REGION Network 9: DataIn - Sollevatore 3
   RUNG wire#powerrail
      "ValveMachine_PB_Connector"(Enable := wire#w1, HMI_PB := "A03_HMI".MB3.Button.A0302.Centratori.Sollevamento, LB_PB_Rest := FALSE, LB_PB_Work := FALSE, LB_PB_StartStop := FALSE, Other_PB := "A03_HMI".MB3.Button.PB_Empty.Valve, PB => "A0302_Centratori".Sollevamento[3].DataIn.PB)
   END_RUNG
   RUNG wire#powerrail
      Contact( "A0302_Centratori".HMI.Selection.Sollevamento[3] )
   END_RUNG wire#w1
   RUNG wire#powerrail
      Contact( "A0302_Centratori_Centraggio_3_Testa_Ls_Basso" )
      Coil( "A0302_Centratori".Sollevamento[3].DataIn.Rest_Ls[1] )
   END_RUNG
   RUNG wire#powerrail
      Contact( "A0302_Centratori_Centraggio_3_Testa_Ls_Alto" )
      Coil( "A0302_Centratori".Sollevamento[3].DataIn.Work_Ls[1] )
   END_RUNG
   // the same network as SCL:
   "ValveMachine_PB_Connector"(Enable := "A0302_Centratori".HMI.Selection.Sollevamento[3],
                           HMI_PB := "A03_HMI".MB3.Button.A0302.Centratori.Sollevamento,
                           LB_PB_Rest := FALSE,
                           LB_PB_Work := FALSE,
                           LB_PB_StartStop := FALSE,
                           Other_PB := "A03_HMI".MB3.Button.PB_Empty.Valve,
                           PB => "A0302_Centratori".Sollevamento[3].DataIn.PB);
   "A0302_Centratori".Sollevamento[3].DataIn.Rest_Ls[1] := "A0302_Centratori_Centraggio_3_Testa_Ls_Basso";
   "A0302_Centratori".Sollevamento[3].DataIn.Work_Ls[1] := "A0302_Centratori_Centraggio_3_Testa_Ls_Alto";
END_REGION

REGION Network 11 (SCL): DSI
   // Di solito facciamo struct DSI con dentro Centratori

   "A0302_Centratori".DSI := "F_DB".DSI_V_Air_A0302_A0303;
END_REGION

REGION Network 12: [Centratori] - Machine Call
   RUNG wire#powerrail
      "A0302_Centratori"(AreaInterface := "Area03".AreaInterface, ZSI := "F_DB".ZSI_Zone25, DSI :=, DataIn :=, CIn :=, Config := "PrjConfig_A03".A0302.Centratori, MachineInterface =>, COut =>)
   END_RUNG
   // the same network as SCL:
   "A0302_Centratori"(AreaInterface := "Area03".AreaInterface,   // "A0302_Centratori_FB"
                      ZSI := "F_DB".ZSI_Zone25,
                      Config := "PrjConfig_A03".A0302.Centratori);
END_REGION

REGION Network 14: <<< DATA OUT >>>
END_REGION

REGION Network 15: DataOut - Centraggio 1
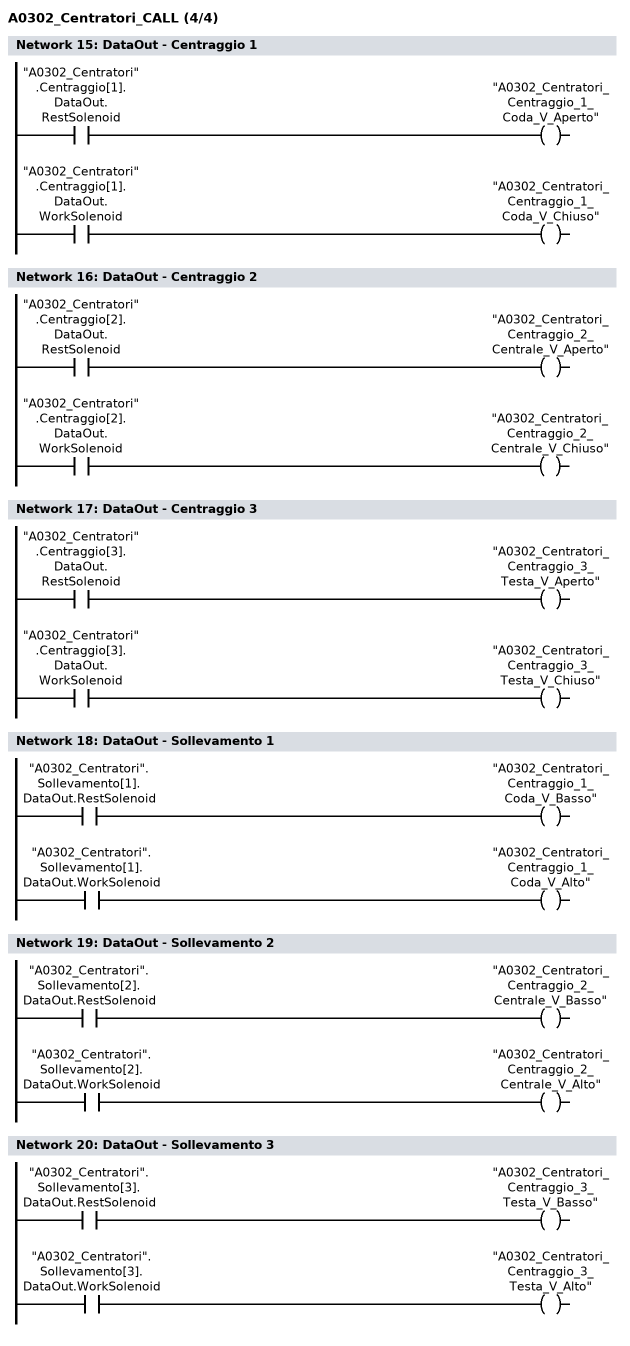
   RUNG wire#powerrail
      Contact( "A0302_Centratori".Centraggio[1].DataOut.RestSolenoid )
      Coil( "A0302_Centratori_Centraggio_1_Coda_V_Aperto" )
   END_RUNG
   RUNG wire#powerrail
      Contact( "A0302_Centratori".Centraggio[1].DataOut.WorkSolenoid )
      Coil( "A0302_Centratori_Centraggio_1_Coda_V_Chiuso" )
   END_RUNG
   // the same network as SCL:
   "A0302_Centratori_Centraggio_1_Coda_V_Aperto" := "A0302_Centratori".Centraggio[1].DataOut.RestSolenoid;
   "A0302_Centratori_Centraggio_1_Coda_V_Chiuso" := "A0302_Centratori".Centraggio[1].DataOut.WorkSolenoid;
END_REGION

REGION Network 16: DataOut - Centraggio 2
   RUNG wire#powerrail
      Contact( "A0302_Centratori".Centraggio[2].DataOut.RestSolenoid )
      Coil( "A0302_Centratori_Centraggio_2_Centrale_V_Aperto" )
   END_RUNG
   RUNG wire#powerrail
      Contact( "A0302_Centratori".Centraggio[2].DataOut.WorkSolenoid )
      Coil( "A0302_Centratori_Centraggio_2_Centrale_V_Chiuso" )
   END_RUNG
   // the same network as SCL:
   "A0302_Centratori_Centraggio_2_Centrale_V_Aperto" := "A0302_Centratori".Centraggio[2].DataOut.RestSolenoid;
   "A0302_Centratori_Centraggio_2_Centrale_V_Chiuso" := "A0302_Centratori".Centraggio[2].DataOut.WorkSolenoid;
END_REGION

REGION Network 17: DataOut - Centraggio 3
   RUNG wire#powerrail
      Contact( "A0302_Centratori".Centraggio[3].DataOut.RestSolenoid )
      Coil( "A0302_Centratori_Centraggio_3_Testa_V_Aperto" )
   END_RUNG
   RUNG wire#powerrail
      Contact( "A0302_Centratori".Centraggio[3].DataOut.WorkSolenoid )
      Coil( "A0302_Centratori_Centraggio_3_Testa_V_Chiuso" )
   END_RUNG
   // the same network as SCL:
   "A0302_Centratori_Centraggio_3_Testa_V_Aperto" := "A0302_Centratori".Centraggio[3].DataOut.RestSolenoid;
   "A0302_Centratori_Centraggio_3_Testa_V_Chiuso" := "A0302_Centratori".Centraggio[3].DataOut.WorkSolenoid;
END_REGION

REGION Network 18: DataOut - Sollevamento 1
   RUNG wire#powerrail
      Contact( "A0302_Centratori".Sollevamento[1].DataOut.RestSolenoid )
      Coil( "A0302_Centratori_Centraggio_1_Coda_V_Basso" )
   END_RUNG
   RUNG wire#powerrail
      Contact( "A0302_Centratori".Sollevamento[1].DataOut.WorkSolenoid )
      Coil( "A0302_Centratori_Centraggio_1_Coda_V_Alto" )
   END_RUNG
   // the same network as SCL:
   "A0302_Centratori_Centraggio_1_Coda_V_Basso" := "A0302_Centratori".Sollevamento[1].DataOut.RestSolenoid;
   "A0302_Centratori_Centraggio_1_Coda_V_Alto" := "A0302_Centratori".Sollevamento[1].DataOut.WorkSolenoid;
END_REGION

REGION Network 19: DataOut - Sollevamento 2
   RUNG wire#powerrail
      Contact( "A0302_Centratori".Sollevamento[2].DataOut.RestSolenoid )
      Coil( "A0302_Centratori_Centraggio_2_Centrale_V_Basso" )
   END_RUNG
   RUNG wire#powerrail
      Contact( "A0302_Centratori".Sollevamento[2].DataOut.WorkSolenoid )
      Coil( "A0302_Centratori_Centraggio_2_Centrale_V_Alto" )
   END_RUNG
   // the same network as SCL:
   "A0302_Centratori_Centraggio_2_Centrale_V_Basso" := "A0302_Centratori".Sollevamento[2].DataOut.RestSolenoid;
   "A0302_Centratori_Centraggio_2_Centrale_V_Alto" := "A0302_Centratori".Sollevamento[2].DataOut.WorkSolenoid;
END_REGION

REGION Network 20: DataOut - Sollevamento 3
   RUNG wire#powerrail
      Contact( "A0302_Centratori".Sollevamento[3].DataOut.RestSolenoid )
      Coil( "A0302_Centratori_Centraggio_3_Testa_V_Basso" )
   END_RUNG
   RUNG wire#powerrail
      Contact( "A0302_Centratori".Sollevamento[3].DataOut.WorkSolenoid )
      Coil( "A0302_Centratori_Centraggio_3_Testa_V_Alto" )
   END_RUNG
   // the same network as SCL:
   "A0302_Centratori_Centraggio_3_Testa_V_Basso" := "A0302_Centratori".Sollevamento[3].DataOut.RestSolenoid;
   "A0302_Centratori_Centraggio_3_Testa_V_Alto" := "A0302_Centratori".Sollevamento[3].DataOut.WorkSolenoid;
END_REGION
END_FUNCTION

FUNCTION_BLOCK "A0302_Centratori_FB"   // FB92, LAD
TITLE = <<< GESTIONE CENTRATORI >>>
// stored: MemoryReserve 100, SetENOAutomatically false
   VAR_INPUT
      AreaInterface : "AreaInterface";
      ZSI : "udt_ZoneSafetyInterface";
      DSI : "udt_DeviceSafetyInterface";
      DataIn : Struct
         OP : "OP_PB";
      END_STRUCT;
      CIn : Struct
         Manager : Struct
            Sollevamento : "ValveMachine_Manager";
            Centraggio : "ValveMachine_Manager";
         END_STRUCT;
         SemiAut_Pb : Bool;
         Rulliera : Struct
            Coda : Struct
               Sens : Struct
                  FTC_Rall : Bool;   // Sensori presenza materiale banco rallentamento ingresso
                  FTC_Prox_Ing : Bool;   // Sensori presenza materiale banco limite ingresso
               END_STRUCT;
            END_STRUCT;
            Centro : Struct
               Sens : Struct
                  FTC_Centrale : Bool;   // 2010BF1 - I50.2
               END_STRUCT;
            END_STRUCT;
         END_STRUCT;
         CarroPareggCoda : Struct
            Ax : "Positioning_DOL_Machine_COut";
            Bloccaggio : "ValveMachine_COut";
            BattutaVerticale : "ValveMachine_COut";
            PareggiatoreLong : "ValveMachine_COut";
            Sens : Struct
               FTC_Ingombro_In : Bool;   // 2012BF1 - I50.0
               FTC_Ingombro_Out : Bool;   // 2012BF2 - I50.1
               PresenzaMat : Bool;   // FC presenza materiale agganciato lato paregg coda
            END_STRUCT;
         END_STRUCT;
         CarroPareggTesta : Struct
            Ax : "Positioning_DOL_Machine_COut";
            Bloccaggio : "ValveMachine_COut";
            Centraggio : "ValveMachine_COut";
            Sollevatore : "ValveMachine_COut";
            Sens : Struct
               FTC1_Rall : Bool;   // 2010BF2 - I50.3
               FTC2_Prox_Ls : Bool;   // 2010BF3 - I50.4
               PresenzaMat : Bool;   // FC presenza materiale agganciato lato paregg testa
            END_STRUCT;
         END_STRUCT;
         BTrk : Struct
            ZoneA0302Entry_Empty : Bool;
            ZoneA0302Exit_Empty : Bool;
         END_STRUCT;
      END_STRUCT;
      Config : Struct
         Centraggio : Array[1..3] of "ValveMachine_Config";
         Sollevamento : Array[1..3] of "ValveMachine_Config";
         DelayMissingCondition : Time;
         WorkWindows : Struct   // Finestre di disattivazione Centratore 1 e 3 in funzione dei Carri
            Coda : Struct
               Min : LReal;
               Max : LReal;
            END_STRUCT;
            Testa : Struct
               Min : LReal;
               Max : LReal;
            END_STRUCT;
         END_STRUCT;
      END_STRUCT;
   END_VAR
   VAR_OUTPUT
      MachineInterface : "MachineInterface";
      COut : Struct
         Centratori : "ValveMachine_COut";
         Centraggio : "ValveMachine_COut";
         Sollevamento : "ValveMachine_COut";
      END_STRUCT;
   END_VAR
   VAR
      Alarm : Struct
         Centraggio : Array[1..3] of "ValveAlr";
         Sollevamento : Array[1..3] of "ValveAlr";
      END_STRUCT;
      Warning : Struct
         Centratore : Array[1..3] of "ValveMachine_Wng";
         Sollevamento : Array[1..3] of "ValveMachine_Wng";
         OP_REST_Centr_MissingCnd : Bool;   // Mancanza comando arresto
         OP_WORK_Centr_MissingCnd : Bool;   // Mancanza consenso lavoro
         OP_REST_Sollev_MissingCnd : Bool;   // Mancanza comando arresto
         OP_WORK_Sollev_MissingCnd : Bool;   // Mancanza consenso lavoro
      END_STRUCT;
      HMI : Struct
         Selection : Struct   // 0=Disable / 1=Enable Pin
            Centraggio : Array[1..3] of Bool;
            Sollevamento : Array[1..3] of Bool;
         END_STRUCT;
         Centratori_Sts : "UDT_HMI-Sts_ValvePosA0301";
         Centraggio_Sts { S7_SetPoint := 'True'} : "UDT_HMI-Sts_ValvePosA0301";
         Sollevamento_Sts { S7_SetPoint := 'True'} : "UDT_HMI-Sts_ValvePosA0301";
      END_STRUCT;
      Centraggio : Array[1..3] of "ValveMachine_FB";
      Sollevamento { S7_SetPoint := 'True'} : Array[1..3] of "ValveMachine_FB";
      Sts : Struct
         Centraggio : Struct
            OP_Rest_Cnd : Bool;
            Op_Work_Cnd : Bool;
         END_STRUCT;
         Sollevamento : Struct
            OP_Rest_Cnd : Bool;
            Op_Work_Cnd : Bool;
         END_STRUCT;
         Centratori_Alarm : Bool;
         Centraggio_AlarmPresence : Bool;
         Sollevamento_AlarmPresence : Bool;
         OP_CanMoveFreely : Bool;
      END_STRUCT;
      Ctrl : Struct
         Centraggio : Struct
            OP_Rest_Man : Bool;
            OP_Work_Man : Bool;
            OP_Rest_Aut : Bool;
            OP_Work_Aut : Bool;
            OP_Rest : Bool;
            OP_Work : Bool;
         END_STRUCT;
         Sollevamento : Struct
            OP_Rest_Man : Bool;
            OP_Work_Man : Bool;
            OP_Rest_Aut : Bool;
            OP_Work_Aut : Bool;
            OP_Rest : Bool;
            OP_Work : Bool;
         END_STRUCT;
      END_STRUCT;
      AUX : Struct
         Centraggio : Struct
            OP_Rest_PB : Bool;
            OP_Work_PB : Bool;
         END_STRUCT;
         Sollevamento : Struct
            OP_Rest_PB : Bool;
            OP_Work_PB : Bool;
         END_STRUCT;
      END_STRUCT;
      TON_OP_REST_Centr_MissingCnd { S7_SetPoint := 'True'} : TON_TIME;
      TON_OP_WORK_Centr_MissingCnd { S7_SetPoint := 'True'} : TON_TIME;
      TON_OP_REST_Sollev_MissingCnd { S7_SetPoint := 'True'} : TON_TIME;
      TON_OP_WORK_Sollev_MissingCnd { S7_SetPoint := 'True'} : TON_TIME;
      DelayMissingCondition : Time;
      TON_Anticipi : Struct
         Work : Struct
            Sollevamento : Array[1..3] of IEC_TIMER;
            Centraggio : Array[1..3] of IEC_TIMER;
         END_STRUCT;
         Rest : Struct
            Sollevamento : Array[1..3] of IEC_TIMER;
            Centraggio : Array[1..3] of IEC_TIMER;
         END_STRUCT;
      END_STRUCT;
   END_VAR
   VAR_TEMP
      PE : Struct
         Centraggio : Struct
            OP_Rest_PB : Bool;
            OP_Work_PB : Bool;
         END_STRUCT;
         Sollevamento : Struct
            OP_Rest_PB : Bool;
            OP_Work_PB : Bool;
         END_STRUCT;
      END_STRUCT;
   END_VAR
   // // Centraggio[1] : Centraggio 1 Coda
   // // Centraggio[2] : Centraggio 2 Centrale
   // // Centraggio[3] : Centraggio 3 Testa
   VAR_TEMP   // added for the SCL form of the ladder/FBD networks
      _w1 : Bool;
      _w2 : Bool;
      _w3 : Bool;
   END_VAR
BEGIN

REGION Network 1: Anticipi Movimento LAVORO
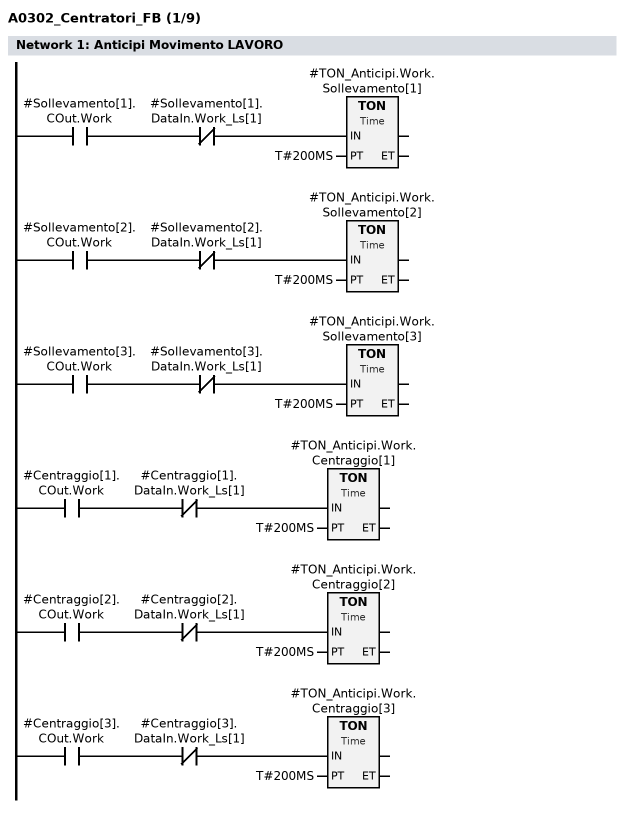
   RUNG wire#powerrail
      Contact( #Sollevamento[1].COut.Work )
      I_Contact( #Sollevamento[1].DataIn.Work_Ls[1] )
      { S7_Templates := "time_type := Time" } #TON_Anticipi.Work.Sollevamento[1].TON(pt := T#200MS, et =>)
   END_RUNG
   RUNG wire#powerrail
      Contact( #Sollevamento[2].COut.Work )
      I_Contact( #Sollevamento[2].DataIn.Work_Ls[1] )
      { S7_Templates := "time_type := Time" } #TON_Anticipi.Work.Sollevamento[2].TON(pt := T#200MS, et =>)
   END_RUNG
   RUNG wire#powerrail
      Contact( #Sollevamento[3].COut.Work )
      I_Contact( #Sollevamento[3].DataIn.Work_Ls[1] )
      { S7_Templates := "time_type := Time" } #TON_Anticipi.Work.Sollevamento[3].TON(pt := T#200MS, et =>)
   END_RUNG
   RUNG wire#powerrail
      Contact( #Centraggio[1].COut.Work )
      I_Contact( #Centraggio[1].DataIn.Work_Ls[1] )
      { S7_Templates := "time_type := Time" } #TON_Anticipi.Work.Centraggio[1].TON(pt := T#200MS, et =>)
   END_RUNG
   RUNG wire#powerrail
      Contact( #Centraggio[2].COut.Work )
      I_Contact( #Centraggio[2].DataIn.Work_Ls[1] )
      { S7_Templates := "time_type := Time" } #TON_Anticipi.Work.Centraggio[2].TON(pt := T#200MS, et =>)
   END_RUNG
   RUNG wire#powerrail
      Contact( #Centraggio[3].COut.Work )
      I_Contact( #Centraggio[3].DataIn.Work_Ls[1] )
      { S7_Templates := "time_type := Time" } #TON_Anticipi.Work.Centraggio[3].TON(pt := T#200MS, et =>)
   END_RUNG
   // the same network as SCL:
   #TON_Anticipi.Work.Sollevamento[1].TON(IN := #Sollevamento[1].COut.Work AND NOT #Sollevamento[1].DataIn.Work_Ls[1],
                           PT := T#200MS);
   #TON_Anticipi.Work.Sollevamento[2].TON(IN := #Sollevamento[2].COut.Work AND NOT #Sollevamento[2].DataIn.Work_Ls[1],
                           PT := T#200MS);
   #TON_Anticipi.Work.Sollevamento[3].TON(IN := #Sollevamento[3].COut.Work AND NOT #Sollevamento[3].DataIn.Work_Ls[1],
                           PT := T#200MS);
   #TON_Anticipi.Work.Centraggio[1].TON(IN := #Centraggio[1].COut.Work AND NOT #Centraggio[1].DataIn.Work_Ls[1],
                           PT := T#200MS);
   #TON_Anticipi.Work.Centraggio[2].TON(IN := #Centraggio[2].COut.Work AND NOT #Centraggio[2].DataIn.Work_Ls[1],
                           PT := T#200MS);
   #TON_Anticipi.Work.Centraggio[3].TON(IN := #Centraggio[3].COut.Work AND NOT #Centraggio[3].DataIn.Work_Ls[1],
                           PT := T#200MS);
END_REGION

REGION Network 2: Anticipi Movimento RIPOSO
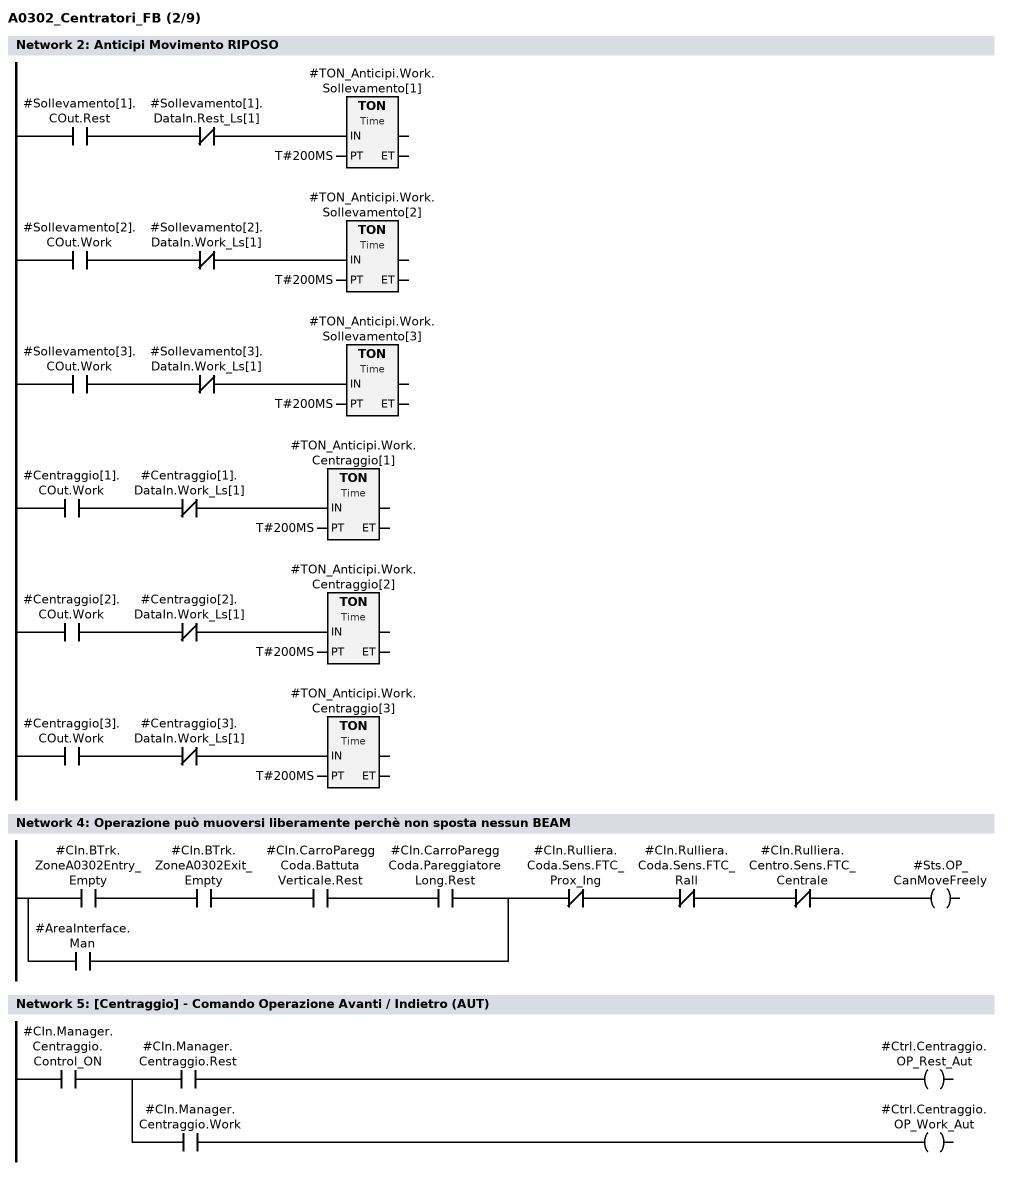
   RUNG wire#powerrail
      Contact( #Sollevamento[1].COut.Rest )
      I_Contact( #Sollevamento[1].DataIn.Rest_Ls[1] )
      { S7_Templates := "time_type := Time" } #TON_Anticipi.Work.Sollevamento[1].TON(pt := T#200MS, et =>)
   END_RUNG
   RUNG wire#powerrail
      Contact( #Sollevamento[2].COut.Work )
      I_Contact( #Sollevamento[2].DataIn.Work_Ls[1] )
      { S7_Templates := "time_type := Time" } #TON_Anticipi.Work.Sollevamento[2].TON(pt := T#200MS, et =>)
   END_RUNG
   RUNG wire#powerrail
      Contact( #Sollevamento[3].COut.Work )
      I_Contact( #Sollevamento[3].DataIn.Work_Ls[1] )
      { S7_Templates := "time_type := Time" } #TON_Anticipi.Work.Sollevamento[3].TON(pt := T#200MS, et =>)
   END_RUNG
   RUNG wire#powerrail
      Contact( #Centraggio[1].COut.Work )
      I_Contact( #Centraggio[1].DataIn.Work_Ls[1] )
      { S7_Templates := "time_type := Time" } #TON_Anticipi.Work.Centraggio[1].TON(pt := T#200MS, et =>)
   END_RUNG
   RUNG wire#powerrail
      Contact( #Centraggio[2].COut.Work )
      I_Contact( #Centraggio[2].DataIn.Work_Ls[1] )
      { S7_Templates := "time_type := Time" } #TON_Anticipi.Work.Centraggio[2].TON(pt := T#200MS, et =>)
   END_RUNG
   RUNG wire#powerrail
      Contact( #Centraggio[3].COut.Work )
      I_Contact( #Centraggio[3].DataIn.Work_Ls[1] )
      { S7_Templates := "time_type := Time" } #TON_Anticipi.Work.Centraggio[3].TON(pt := T#200MS, et =>)
   END_RUNG
   // the same network as SCL:
   #TON_Anticipi.Work.Sollevamento[1].TON(IN := #Sollevamento[1].COut.Rest AND NOT #Sollevamento[1].DataIn.Rest_Ls[1],
                           PT := T#200MS);
   #TON_Anticipi.Work.Sollevamento[2].TON(IN := #Sollevamento[2].COut.Work AND NOT #Sollevamento[2].DataIn.Work_Ls[1],
                           PT := T#200MS);
   #TON_Anticipi.Work.Sollevamento[3].TON(IN := #Sollevamento[3].COut.Work AND NOT #Sollevamento[3].DataIn.Work_Ls[1],
                           PT := T#200MS);
   #TON_Anticipi.Work.Centraggio[1].TON(IN := #Centraggio[1].COut.Work AND NOT #Centraggio[1].DataIn.Work_Ls[1],
                           PT := T#200MS);
   #TON_Anticipi.Work.Centraggio[2].TON(IN := #Centraggio[2].COut.Work AND NOT #Centraggio[2].DataIn.Work_Ls[1],
                           PT := T#200MS);
   #TON_Anticipi.Work.Centraggio[3].TON(IN := #Centraggio[3].COut.Work AND NOT #Centraggio[3].DataIn.Work_Ls[1],
                           PT := T#200MS);
END_REGION

REGION Network 3: <+>
END_REGION

REGION Network 4: Operazione può muoversi liberamente perchè non sposta nessun BEAM
   RUNG wire#powerrail
      Contact( #CIn.BTrk.ZoneA0302Entry_Empty )
      Contact( #CIn.BTrk.ZoneA0302Exit_Empty )
      Contact( #CIn.CarroPareggCoda.BattutaVerticale.Rest )
      Contact( #CIn.CarroPareggCoda.PareggiatoreLong.Rest )
      wire#w1
      I_Contact( #CIn.Rulliera.Coda.Sens.FTC_Prox_Ing )
      I_Contact( #CIn.Rulliera.Coda.Sens.FTC_Rall )
      I_Contact( #CIn.Rulliera.Centro.Sens.FTC_Centrale )
      Coil( #Sts.OP_CanMoveFreely )
   END_RUNG
   RUNG wire#powerrail
      Contact( #AreaInterface.Man )
   END_RUNG wire#w1
   // the same network as SCL:
   #Sts.OP_CanMoveFreely := ((#CIn.BTrk.ZoneA0302Entry_Empty AND #CIn.BTrk.ZoneA0302Exit_Empty AND #CIn.CarroPareggCoda.BattutaVerticale.Rest AND #CIn.CarroPareggCoda.PareggiatoreLong.Rest) OR #AreaInterface.Man) AND NOT #CIn.Rulliera.Coda.Sens.FTC_Prox_Ing AND NOT #CIn.Rulliera.Coda.Sens.FTC_Rall AND NOT #CIn.Rulliera.Centro.Sens.FTC_Centrale;
END_REGION

REGION Network 5: [Centraggio] - Comando Operazione Avanti / Indietro (AUT)
   RUNG wire#powerrail
      Contact( #CIn.Manager.Centraggio.Control_ON )
      wire#w1
      Contact( #CIn.Manager.Centraggio.Rest )
      Coil( #Ctrl.Centraggio.OP_Rest_Aut )
   END_RUNG
   RUNG wire#w1
      Contact( #CIn.Manager.Centraggio.Work )
      Coil( #Ctrl.Centraggio.OP_Work_Aut )
   END_RUNG
   // the same network as SCL:
   #Ctrl.Centraggio.OP_Rest_Aut := #CIn.Manager.Centraggio.Control_ON AND #CIn.Manager.Centraggio.Rest;
   #Ctrl.Centraggio.OP_Work_Aut := #CIn.Manager.Centraggio.Control_ON AND #CIn.Manager.Centraggio.Work;
END_REGION

REGION Network 6: [Centraggio] - Comando Operazione Lavoro / Riposo (MAN)
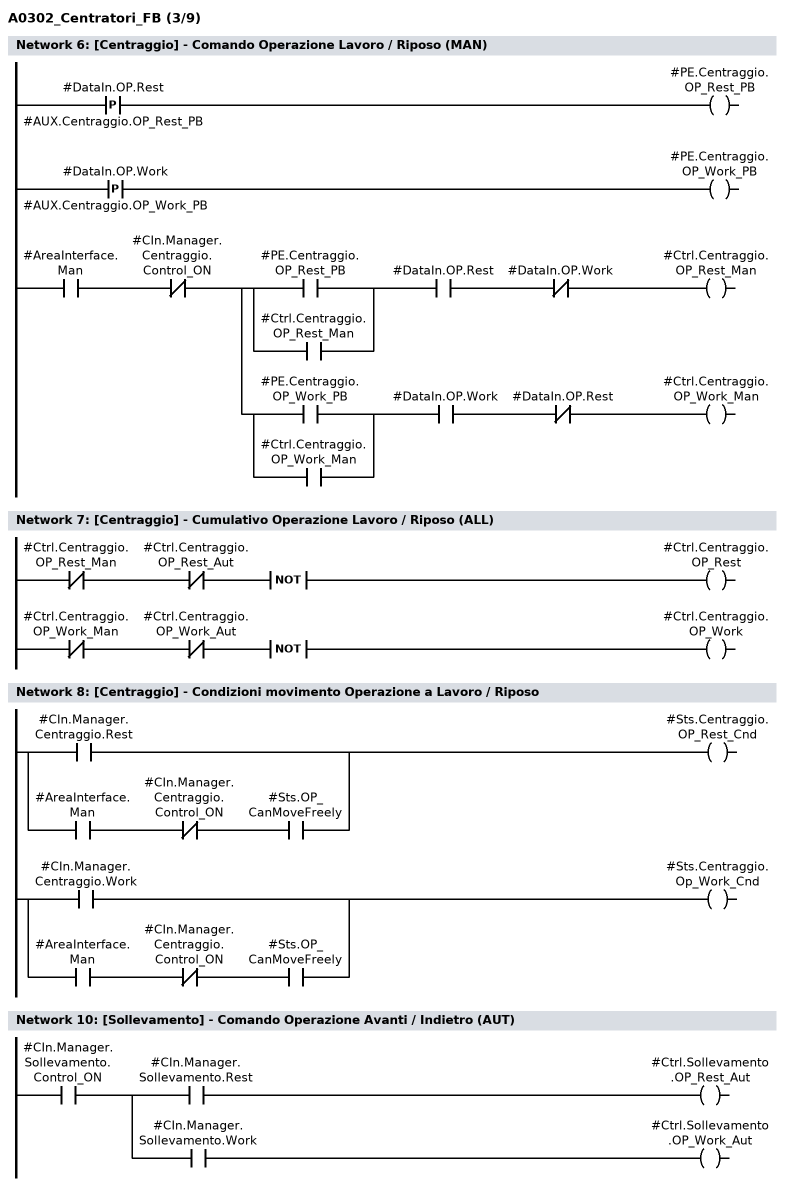
   RUNG wire#powerrail
      P_Contact(operand := #DataIn.OP.Rest, bit := #AUX.Centraggio.OP_Rest_PB)
      Coil( #PE.Centraggio.OP_Rest_PB )
   END_RUNG
   RUNG wire#powerrail
      P_Contact(operand := #DataIn.OP.Work, bit := #AUX.Centraggio.OP_Work_PB)
      Coil( #PE.Centraggio.OP_Work_PB )
   END_RUNG
   RUNG wire#powerrail
      Contact( #AreaInterface.Man )
      I_Contact( #CIn.Manager.Centraggio.Control_ON )
      wire#w1
      Contact( #PE.Centraggio.OP_Rest_PB )
      wire#w2
      Contact( #DataIn.OP.Rest )
      I_Contact( #DataIn.OP.Work )
      Coil( #Ctrl.Centraggio.OP_Rest_Man )
   END_RUNG
   RUNG wire#w1
      Contact( #Ctrl.Centraggio.OP_Rest_Man )
   END_RUNG wire#w2
   RUNG wire#w1
      Contact( #PE.Centraggio.OP_Work_PB )
      wire#w3
      Contact( #DataIn.OP.Work )
      I_Contact( #DataIn.OP.Rest )
      Coil( #Ctrl.Centraggio.OP_Work_Man )
   END_RUNG
   RUNG wire#w1
      Contact( #Ctrl.Centraggio.OP_Work_Man )
   END_RUNG wire#w3
   // the same network as SCL:
   #_w1 := #DataIn.OP.Rest AND NOT #AUX.Centraggio.OP_Rest_PB;   // rising edge of #DataIn.OP.Rest
   #AUX.Centraggio.OP_Rest_PB := #DataIn.OP.Rest;
   #PE.Centraggio.OP_Rest_PB := #_w1;
   #_w2 := #DataIn.OP.Work AND NOT #AUX.Centraggio.OP_Work_PB;   // rising edge of #DataIn.OP.Work
   #AUX.Centraggio.OP_Work_PB := #DataIn.OP.Work;
   #PE.Centraggio.OP_Work_PB := #_w2;
   #_w3 := #AreaInterface.Man AND NOT #CIn.Manager.Centraggio.Control_ON;
   #Ctrl.Centraggio.OP_Rest_Man := #_w3 AND (#PE.Centraggio.OP_Rest_PB OR #Ctrl.Centraggio.OP_Rest_Man) AND #DataIn.OP.Rest AND NOT #DataIn.OP.Work;
   #Ctrl.Centraggio.OP_Work_Man := #_w3 AND (#PE.Centraggio.OP_Work_PB OR #Ctrl.Centraggio.OP_Work_Man) AND #DataIn.OP.Work AND NOT #DataIn.OP.Rest;
END_REGION

REGION Network 7: [Centraggio] - Cumulativo Operazione Lavoro / Riposo (ALL)
   RUNG wire#powerrail
      I_Contact( #Ctrl.Centraggio.OP_Rest_Man )
      I_Contact( #Ctrl.Centraggio.OP_Rest_Aut )
      Not()
      Coil( #Ctrl.Centraggio.OP_Rest )
   END_RUNG
   RUNG wire#powerrail
      I_Contact( #Ctrl.Centraggio.OP_Work_Man )
      I_Contact( #Ctrl.Centraggio.OP_Work_Aut )
      Not()
      Coil( #Ctrl.Centraggio.OP_Work )
   END_RUNG
   // the same network as SCL:
   #Ctrl.Centraggio.OP_Rest := NOT (NOT #Ctrl.Centraggio.OP_Rest_Man AND NOT #Ctrl.Centraggio.OP_Rest_Aut);
   #Ctrl.Centraggio.OP_Work := NOT (NOT #Ctrl.Centraggio.OP_Work_Man AND NOT #Ctrl.Centraggio.OP_Work_Aut);
END_REGION

REGION Network 8: [Centraggio] - Condizioni movimento Operazione a Lavoro / Riposo
   RUNG wire#powerrail
      Contact( #CIn.Manager.Centraggio.Rest )
      wire#w1
      Coil( #Sts.Centraggio.OP_Rest_Cnd )
   END_RUNG
   RUNG wire#powerrail
      Contact( #AreaInterface.Man )
      I_Contact( #CIn.Manager.Centraggio.Control_ON )
      Contact( #Sts.OP_CanMoveFreely )
   END_RUNG wire#w1
   RUNG wire#powerrail
      Contact( #CIn.Manager.Centraggio.Work )
      wire#w2
      Coil( #Sts.Centraggio.Op_Work_Cnd )
   END_RUNG
   RUNG wire#powerrail
      Contact( #AreaInterface.Man )
      I_Contact( #CIn.Manager.Centraggio.Control_ON )
      Contact( #Sts.OP_CanMoveFreely )
   END_RUNG wire#w2
   // the same network as SCL:
   #Sts.Centraggio.OP_Rest_Cnd := #CIn.Manager.Centraggio.Rest OR (#AreaInterface.Man AND NOT #CIn.Manager.Centraggio.Control_ON AND #Sts.OP_CanMoveFreely);
   #Sts.Centraggio.Op_Work_Cnd := #CIn.Manager.Centraggio.Work OR (#AreaInterface.Man AND NOT #CIn.Manager.Centraggio.Control_ON AND #Sts.OP_CanMoveFreely);
END_REGION

REGION Network 10: [Sollevamento] - Comando Operazione Avanti / Indietro (AUT)
   RUNG wire#powerrail
      Contact( #CIn.Manager.Sollevamento.Control_ON )
      wire#w1
      Contact( #CIn.Manager.Sollevamento.Rest )
      Coil( #Ctrl.Sollevamento.OP_Rest_Aut )
   END_RUNG
   RUNG wire#w1
      Contact( #CIn.Manager.Sollevamento.Work )
      Coil( #Ctrl.Sollevamento.OP_Work_Aut )
   END_RUNG
   // the same network as SCL:
   #Ctrl.Sollevamento.OP_Rest_Aut := #CIn.Manager.Sollevamento.Control_ON AND #CIn.Manager.Sollevamento.Rest;
   #Ctrl.Sollevamento.OP_Work_Aut := #CIn.Manager.Sollevamento.Control_ON AND #CIn.Manager.Sollevamento.Work;
END_REGION

REGION Network 11: [Sollevamento] - Comando Operazione Lavoro / Riposo (MAN)
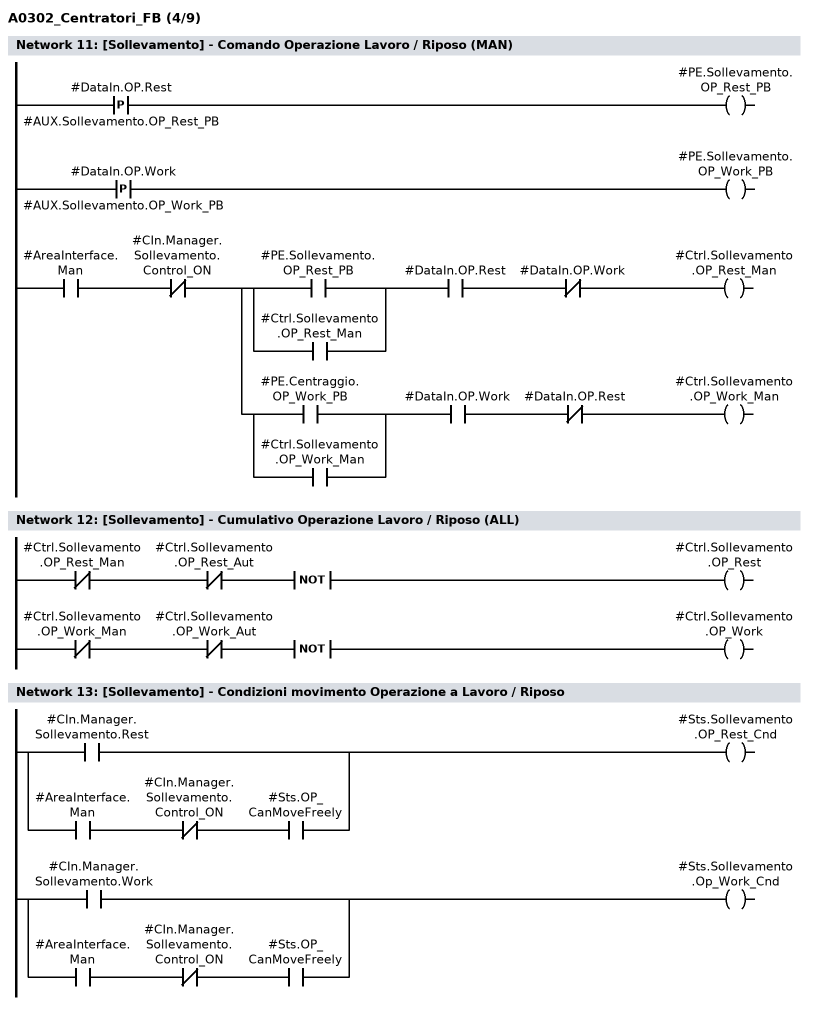
   RUNG wire#powerrail
      P_Contact(operand := #DataIn.OP.Rest, bit := #AUX.Sollevamento.OP_Rest_PB)
      Coil( #PE.Sollevamento.OP_Rest_PB )
   END_RUNG
   RUNG wire#powerrail
      P_Contact(operand := #DataIn.OP.Work, bit := #AUX.Sollevamento.OP_Work_PB)
      Coil( #PE.Sollevamento.OP_Work_PB )
   END_RUNG
   RUNG wire#powerrail
      Contact( #AreaInterface.Man )
      I_Contact( #CIn.Manager.Sollevamento.Control_ON )
      wire#w1
      Contact( #PE.Sollevamento.OP_Rest_PB )
      wire#w2
      Contact( #DataIn.OP.Rest )
      I_Contact( #DataIn.OP.Work )
      Coil( #Ctrl.Sollevamento.OP_Rest_Man )
   END_RUNG
   RUNG wire#w1
      Contact( #Ctrl.Sollevamento.OP_Rest_Man )
   END_RUNG wire#w2
   RUNG wire#w1
      Contact( #PE.Centraggio.OP_Work_PB )
      wire#w3
      Contact( #DataIn.OP.Work )
      I_Contact( #DataIn.OP.Rest )
      Coil( #Ctrl.Sollevamento.OP_Work_Man )
   END_RUNG
   RUNG wire#w1
      Contact( #Ctrl.Sollevamento.OP_Work_Man )
   END_RUNG wire#w3
   // the same network as SCL:
   #_w1 := #DataIn.OP.Rest AND NOT #AUX.Sollevamento.OP_Rest_PB;   // rising edge of #DataIn.OP.Rest
   #AUX.Sollevamento.OP_Rest_PB := #DataIn.OP.Rest;
   #PE.Sollevamento.OP_Rest_PB := #_w1;
   #_w2 := #DataIn.OP.Work AND NOT #AUX.Sollevamento.OP_Work_PB;   // rising edge of #DataIn.OP.Work
   #AUX.Sollevamento.OP_Work_PB := #DataIn.OP.Work;
   #PE.Sollevamento.OP_Work_PB := #_w2;
   #_w3 := #AreaInterface.Man AND NOT #CIn.Manager.Sollevamento.Control_ON;
   #Ctrl.Sollevamento.OP_Rest_Man := #_w3 AND (#PE.Sollevamento.OP_Rest_PB OR #Ctrl.Sollevamento.OP_Rest_Man) AND #DataIn.OP.Rest AND NOT #DataIn.OP.Work;
   #Ctrl.Sollevamento.OP_Work_Man := #_w3 AND (#PE.Centraggio.OP_Work_PB OR #Ctrl.Sollevamento.OP_Work_Man) AND #DataIn.OP.Work AND NOT #DataIn.OP.Rest;
END_REGION

REGION Network 12: [Sollevamento] - Cumulativo Operazione Lavoro / Riposo (ALL)
   RUNG wire#powerrail
      I_Contact( #Ctrl.Sollevamento.OP_Rest_Man )
      I_Contact( #Ctrl.Sollevamento.OP_Rest_Aut )
      Not()
      Coil( #Ctrl.Sollevamento.OP_Rest )
   END_RUNG
   RUNG wire#powerrail
      I_Contact( #Ctrl.Sollevamento.OP_Work_Man )
      I_Contact( #Ctrl.Sollevamento.OP_Work_Aut )
      Not()
      Coil( #Ctrl.Sollevamento.OP_Work )
   END_RUNG
   // the same network as SCL:
   #Ctrl.Sollevamento.OP_Rest := NOT (NOT #Ctrl.Sollevamento.OP_Rest_Man AND NOT #Ctrl.Sollevamento.OP_Rest_Aut);
   #Ctrl.Sollevamento.OP_Work := NOT (NOT #Ctrl.Sollevamento.OP_Work_Man AND NOT #Ctrl.Sollevamento.OP_Work_Aut);
END_REGION

REGION Network 13: [Sollevamento] - Condizioni movimento Operazione a Lavoro / Riposo
   RUNG wire#powerrail
      Contact( #CIn.Manager.Sollevamento.Rest )
      wire#w1
      Coil( #Sts.Sollevamento.OP_Rest_Cnd )
   END_RUNG
   RUNG wire#powerrail
      Contact( #AreaInterface.Man )
      I_Contact( #CIn.Manager.Sollevamento.Control_ON )
      Contact( #Sts.OP_CanMoveFreely )
   END_RUNG wire#w1
   RUNG wire#powerrail
      Contact( #CIn.Manager.Sollevamento.Work )
      wire#w2
      Coil( #Sts.Sollevamento.Op_Work_Cnd )
   END_RUNG
   RUNG wire#powerrail
      Contact( #AreaInterface.Man )
      I_Contact( #CIn.Manager.Sollevamento.Control_ON )
      Contact( #Sts.OP_CanMoveFreely )
   END_RUNG wire#w2
   // the same network as SCL:
   #Sts.Sollevamento.OP_Rest_Cnd := #CIn.Manager.Sollevamento.Rest OR (#AreaInterface.Man AND NOT #CIn.Manager.Sollevamento.Control_ON AND #Sts.OP_CanMoveFreely);
   #Sts.Sollevamento.Op_Work_Cnd := #CIn.Manager.Sollevamento.Work OR (#AreaInterface.Man AND NOT #CIn.Manager.Sollevamento.Control_ON AND #Sts.OP_CanMoveFreely);
END_REGION

REGION Network 15 (SCL): Centraggio + Sollevamento - Cin Manager (Esecuzione sequenza comandi)
   //
   #Centraggio[1].Cin.Manager.Control_ON := #Centraggio[2].Cin.Manager.Control_ON :=
   #Centraggio[3].Cin.Manager.Control_ON := #CIn.Manager.Centraggio.Control_ON;
   //
   #Sollevamento[1].Cin.Manager.Control_ON :=#Sollevamento[2].Cin.Manager.Control_ON :=
   #Sollevamento[3].Cin.Manager.Control_ON := #CIn.Manager.Sollevamento.Control_ON;

   REGION Se nessun comando attivo resetto il comando Work/Rest
       #Centraggio[1].Cin.Manager.Rest := FALSE;
       #Centraggio[2].Cin.Manager.Rest := FALSE;
       #Centraggio[3].Cin.Manager.Rest := FALSE;

       #Centraggio[1].Cin.Manager.Work := FALSE;
       #Centraggio[2].Cin.Manager.Work := FALSE;
       #Centraggio[3].Cin.Manager.Work := FALSE;

       #Sollevamento[1].Cin.Manager.Rest := FALSE;
       #Sollevamento[2].Cin.Manager.Rest := FALSE;
       #Sollevamento[3].Cin.Manager.Rest := FALSE;

       #Sollevamento[1].Cin.Manager.Work := FALSE;
       #Sollevamento[2].Cin.Manager.Work := FALSE;
       #Sollevamento[3].Cin.Manager.Work := FALSE;
   END_REGION ;


   IF #AreaInterface.Aut OR #CIn.SemiAut_Pb THEN

       IF #Ctrl.Sollevamento.OP_Rest AND #Sts.Sollevamento.OP_Rest_Cnd
           AND #Centraggio[2].COut.Rest THEN
           #Sollevamento[1].Cin.Manager.Rest := TRUE;
           #Sollevamento[2].Cin.Manager.Rest := TRUE;
           #Sollevamento[3].Cin.Manager.Rest := TRUE;

       ELSIF #Ctrl.Sollevamento.OP_Work AND #Sts.Sollevamento.Op_Work_Cnd THEN
           #Sollevamento[1].Cin.Manager.Work := TRUE;
           #Sollevamento[2].Cin.Manager.Work := TRUE;
           #Sollevamento[3].Cin.Manager.Work := TRUE;

       END_IF;


       IF #Ctrl.Centraggio.OP_Rest AND #Sts.Centraggio.OP_Rest_Cnd THEN
           #Centraggio[1].Cin.Manager.Rest := TRUE;
           #Centraggio[2].Cin.Manager.Rest := TRUE;
           #Centraggio[3].Cin.Manager.Rest := TRUE;

       ELSIF #Ctrl.Centraggio.OP_Work AND #Sts.Centraggio.Op_Work_Cnd
           AND #Sollevamento[2].COut.Work THEN
           #Centraggio[1].Cin.Manager.Work := TRUE;
           #Centraggio[2].Cin.Manager.Work := TRUE;
           #Centraggio[3].Cin.Manager.Work := TRUE;

       END_IF;
   END_IF;
END_REGION

REGION Network 16 (SCL): Centraggio + Sollevamento - CIn Abilitazioni Manager
   #Centraggio[1].Cin.Manager.EnableStopDoorOpeningReq := #Centraggio[2].Cin.Manager.EnableStopDoorOpeningReq :=
   #Centraggio[3].Cin.Manager.EnableStopDoorOpeningReq := #CIn.Manager.Centraggio.EnableStopDoorOpeningReq;

   #Sollevamento[1].Cin.Manager.EnableStopDoorOpeningReq := #Sollevamento[2].Cin.Manager.EnableStopDoorOpeningReq :=
   #Sollevamento[3].Cin.Manager.EnableStopDoorOpeningReq := #CIn.Manager.Sollevamento.EnableStopDoorOpeningReq;

   #Centraggio[1].Cin.Manager.EnableStopInPhase := #Centraggio[2].Cin.Manager.EnableStopInPhase :=
   #Centraggio[3].Cin.Manager.EnableStopInPhase := #CIn.Manager.Centraggio.EnableStopInPhase;

   #Sollevamento[1].Cin.Manager.EnableStopInPhase :=#Sollevamento[2].Cin.Manager.EnableStopInPhase:=
   #Sollevamento[3].Cin.Manager.EnableStopInPhase:= #CIn.Manager.Sollevamento.EnableStopInPhase;

   #Centraggio[1].Cin.Manager.EnableStopProgrammed := #Centraggio[2].Cin.Manager.EnableStopProgrammed
   := #Centraggio[3].Cin.Manager.EnableStopProgrammed := #CIn.Manager.Centraggio.EnableStopProgrammed;

   #Sollevamento[1].Cin.Manager.EnableStopProgrammed :=#Sollevamento[2].Cin.Manager.EnableStopProgrammed:=
   #Sollevamento[3].Cin.Manager.EnableStopProgrammed:=  #CIn.Manager.Sollevamento.EnableStopProgrammed;
END_REGION

REGION Network 17: <+>
END_REGION

REGION Network 18: [Centraggio] - Warning manacanza condizioni esecuzione Operazione RIPOSO / LAVORO
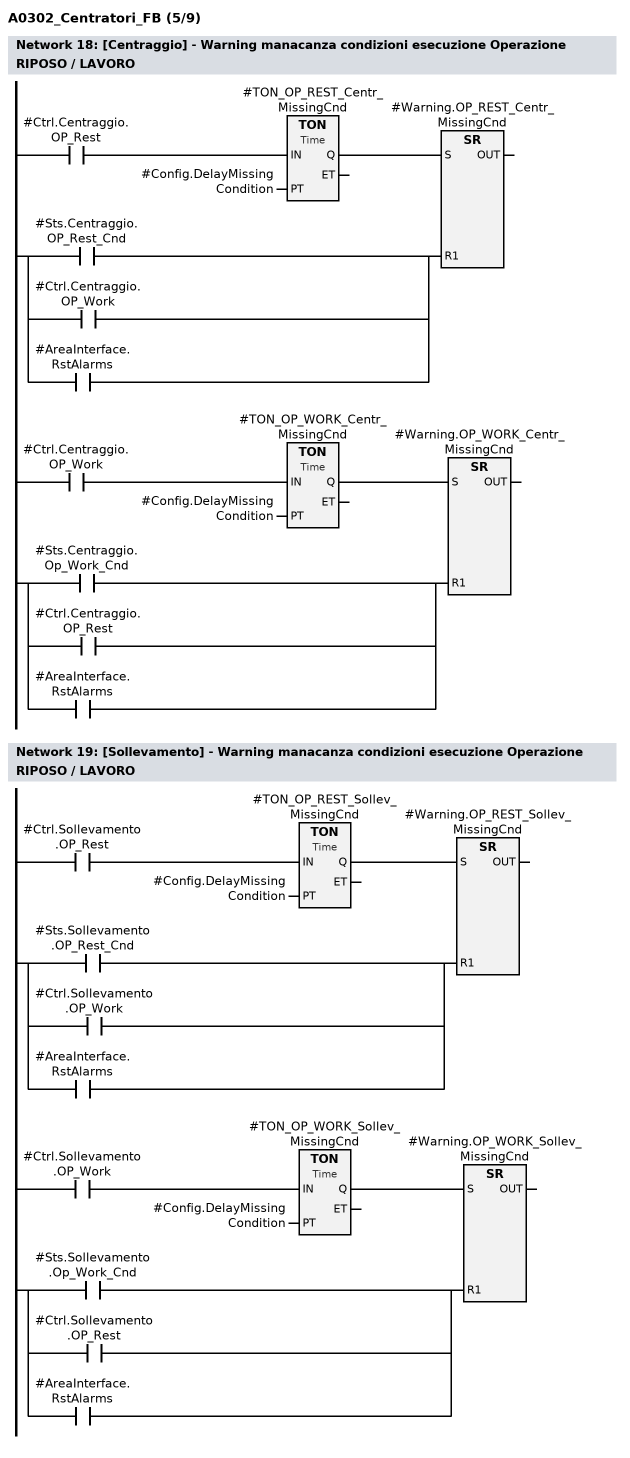
   RUNG wire#powerrail
      Contact( #Ctrl.Centraggio.OP_Rest )
      { S7_Templates := "time_type := Time" } #TON_OP_REST_Centr_MissingCnd.TON(pt := #Config.DelayMissingCondition, et =>)
      S_SR(operand := #Warning.OP_REST_Centr_MissingCnd, r1 := wire#w1)
   END_RUNG
   RUNG wire#powerrail
      Contact( #Sts.Centraggio.OP_Rest_Cnd )
   END_RUNG wire#w1
   RUNG wire#powerrail
      Contact( #Ctrl.Centraggio.OP_Work )
   END_RUNG wire#w1
   RUNG wire#powerrail
      Contact( #AreaInterface.RstAlarms )
   END_RUNG wire#w1
   RUNG wire#powerrail
      Contact( #Ctrl.Centraggio.OP_Work )
      { S7_Templates := "time_type := Time" } #TON_OP_WORK_Centr_MissingCnd.TON(pt := #Config.DelayMissingCondition, et =>)
      S_SR(operand := #Warning.OP_WORK_Centr_MissingCnd, r1 := wire#w2)
   END_RUNG
   RUNG wire#powerrail
      Contact( #Sts.Centraggio.Op_Work_Cnd )
   END_RUNG wire#w2
   RUNG wire#powerrail
      Contact( #Ctrl.Centraggio.OP_Rest )
   END_RUNG wire#w2
   RUNG wire#powerrail
      Contact( #AreaInterface.RstAlarms )
   END_RUNG wire#w2
   // the same network as SCL:
   #TON_OP_REST_Centr_MissingCnd(IN := #Ctrl.Centraggio.OP_Rest, PT := #Config.DelayMissingCondition);   // TON
   IF #TON_OP_REST_Centr_MissingCnd.Q THEN
       #Warning.OP_REST_Centr_MissingCnd := TRUE;   // SR flip-flop
   END_IF;
   IF #Sts.Centraggio.OP_Rest_Cnd OR #Ctrl.Centraggio.OP_Work OR #AreaInterface.RstAlarms THEN
       #Warning.OP_REST_Centr_MissingCnd := FALSE;
   END_IF;
   #TON_OP_WORK_Centr_MissingCnd(IN := #Ctrl.Centraggio.OP_Work, PT := #Config.DelayMissingCondition);   // TON
   IF #TON_OP_WORK_Centr_MissingCnd.Q THEN
       #Warning.OP_WORK_Centr_MissingCnd := TRUE;   // SR flip-flop
   END_IF;
   IF #Sts.Centraggio.Op_Work_Cnd OR #Ctrl.Centraggio.OP_Rest OR #AreaInterface.RstAlarms THEN
       #Warning.OP_WORK_Centr_MissingCnd := FALSE;
   END_IF;
END_REGION

REGION Network 19: [Sollevamento] - Warning manacanza condizioni esecuzione Operazione RIPOSO / LAVORO
   RUNG wire#powerrail
      Contact( #Ctrl.Sollevamento.OP_Rest )
      { S7_Templates := "time_type := Time" } #TON_OP_REST_Sollev_MissingCnd.TON(pt := #Config.DelayMissingCondition, et =>)
      S_SR(operand := #Warning.OP_REST_Sollev_MissingCnd, r1 := wire#w1)
   END_RUNG
   RUNG wire#powerrail
      Contact( #Sts.Sollevamento.OP_Rest_Cnd )
   END_RUNG wire#w1
   RUNG wire#powerrail
      Contact( #Ctrl.Sollevamento.OP_Work )
   END_RUNG wire#w1
   RUNG wire#powerrail
      Contact( #AreaInterface.RstAlarms )
   END_RUNG wire#w1
   RUNG wire#powerrail
      Contact( #Ctrl.Sollevamento.OP_Work )
      { S7_Templates := "time_type := Time" } #TON_OP_WORK_Sollev_MissingCnd.TON(pt := #Config.DelayMissingCondition, et =>)
      S_SR(operand := #Warning.OP_WORK_Sollev_MissingCnd, r1 := wire#w2)
   END_RUNG
   RUNG wire#powerrail
      Contact( #Sts.Sollevamento.Op_Work_Cnd )
   END_RUNG wire#w2
   RUNG wire#powerrail
      Contact( #Ctrl.Sollevamento.OP_Rest )
   END_RUNG wire#w2
   RUNG wire#powerrail
      Contact( #AreaInterface.RstAlarms )
   END_RUNG wire#w2
   // the same network as SCL:
   #TON_OP_REST_Sollev_MissingCnd(IN := #Ctrl.Sollevamento.OP_Rest, PT := #Config.DelayMissingCondition);   // TON
   IF #TON_OP_REST_Sollev_MissingCnd.Q THEN
       #Warning.OP_REST_Sollev_MissingCnd := TRUE;   // SR flip-flop
   END_IF;
   IF #Sts.Sollevamento.OP_Rest_Cnd OR #Ctrl.Sollevamento.OP_Work OR #AreaInterface.RstAlarms THEN
       #Warning.OP_REST_Sollev_MissingCnd := FALSE;
   END_IF;
   #TON_OP_WORK_Sollev_MissingCnd(IN := #Ctrl.Sollevamento.OP_Work, PT := #Config.DelayMissingCondition);   // TON
   IF #TON_OP_WORK_Sollev_MissingCnd.Q THEN
       #Warning.OP_WORK_Sollev_MissingCnd := TRUE;   // SR flip-flop
   END_IF;
   IF #Sts.Sollevamento.Op_Work_Cnd OR #Ctrl.Sollevamento.OP_Rest OR #AreaInterface.RstAlarms THEN
       #Warning.OP_WORK_Sollev_MissingCnd := FALSE;
   END_IF;
END_REGION

REGION Network 21: Centraggio - CIn External alarm
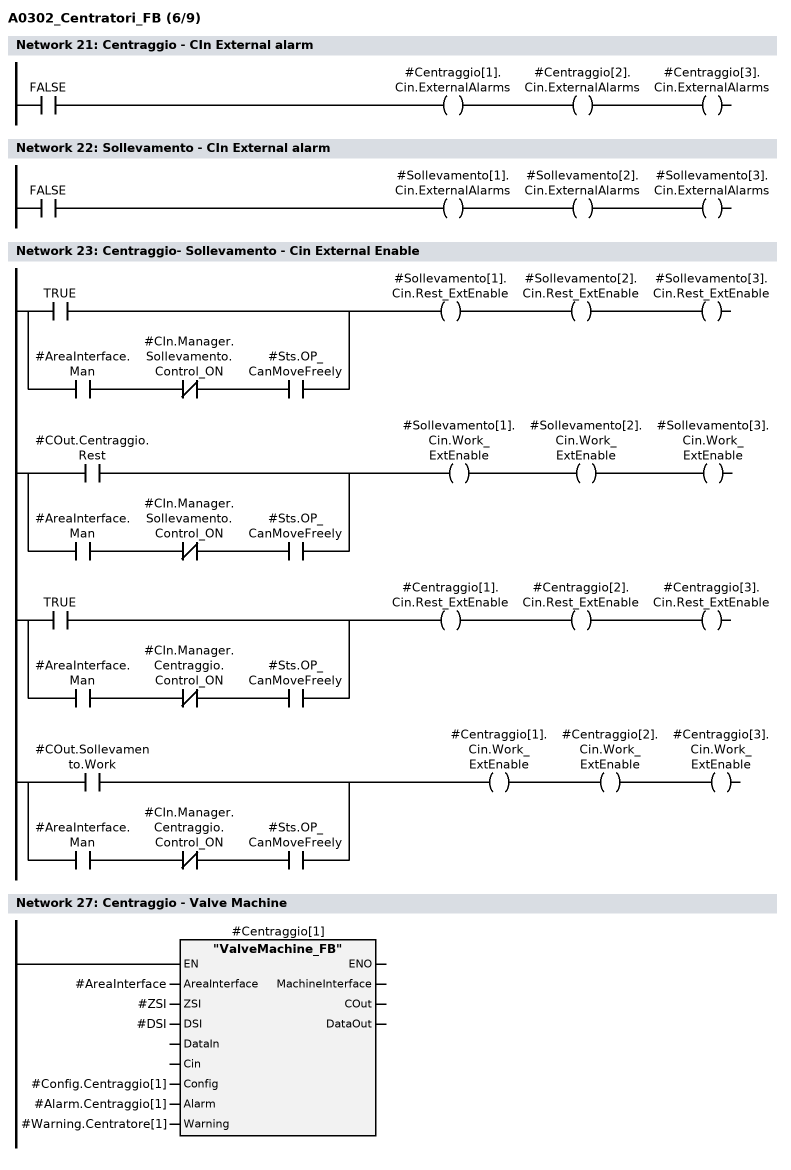
   RUNG wire#powerrail
      Contact( FALSE )
      Coil( #Centraggio[1].Cin.ExternalAlarms )
      Coil( #Centraggio[2].Cin.ExternalAlarms )
      Coil( #Centraggio[3].Cin.ExternalAlarms )
   END_RUNG
   // the same network as SCL:
   #Centraggio[1].Cin.ExternalAlarms := FALSE;
   #Centraggio[2].Cin.ExternalAlarms := FALSE;
   #Centraggio[3].Cin.ExternalAlarms := FALSE;
END_REGION

REGION Network 22: Sollevamento - CIn External alarm
   RUNG wire#powerrail
      Contact( FALSE )
      Coil( #Sollevamento[1].Cin.ExternalAlarms )
      Coil( #Sollevamento[2].Cin.ExternalAlarms )
      Coil( #Sollevamento[3].Cin.ExternalAlarms )
   END_RUNG
   // the same network as SCL:
   #Sollevamento[1].Cin.ExternalAlarms := FALSE;
   #Sollevamento[2].Cin.ExternalAlarms := FALSE;
   #Sollevamento[3].Cin.ExternalAlarms := FALSE;
END_REGION

REGION Network 23: Centraggio- Sollevamento - Cin External Enable
   RUNG wire#powerrail
      Contact( TRUE )
      wire#w1
      Coil( #Sollevamento[1].Cin.Rest_ExtEnable )
      Coil( #Sollevamento[2].Cin.Rest_ExtEnable )
      Coil( #Sollevamento[3].Cin.Rest_ExtEnable )
   END_RUNG
   RUNG wire#powerrail
      Contact( #AreaInterface.Man )
      I_Contact( #CIn.Manager.Sollevamento.Control_ON )
      Contact( #Sts.OP_CanMoveFreely )
   END_RUNG wire#w1
   RUNG wire#powerrail
      Contact( #COut.Centraggio.Rest )
      wire#w2
      Coil( #Sollevamento[1].Cin.Work_ExtEnable )
      Coil( #Sollevamento[2].Cin.Work_ExtEnable )
      Coil( #Sollevamento[3].Cin.Work_ExtEnable )
   END_RUNG
   RUNG wire#powerrail
      Contact( #AreaInterface.Man )
      I_Contact( #CIn.Manager.Sollevamento.Control_ON )
      Contact( #Sts.OP_CanMoveFreely )
   END_RUNG wire#w2
   RUNG wire#powerrail
      Contact( TRUE )
      wire#w3
      Coil( #Centraggio[1].Cin.Rest_ExtEnable )
      Coil( #Centraggio[2].Cin.Rest_ExtEnable )
      Coil( #Centraggio[3].Cin.Rest_ExtEnable )
   END_RUNG
   RUNG wire#powerrail
      Contact( #AreaInterface.Man )
      I_Contact( #CIn.Manager.Centraggio.Control_ON )
      Contact( #Sts.OP_CanMoveFreely )
   END_RUNG wire#w3
   RUNG wire#powerrail
      Contact( #COut.Sollevamento.Work )
      wire#w4
      Coil( #Centraggio[1].Cin.Work_ExtEnable )
      Coil( #Centraggio[2].Cin.Work_ExtEnable )
      Coil( #Centraggio[3].Cin.Work_ExtEnable )
   END_RUNG
   RUNG wire#powerrail
      Contact( #AreaInterface.Man )
      I_Contact( #CIn.Manager.Centraggio.Control_ON )
      Contact( #Sts.OP_CanMoveFreely )
   END_RUNG wire#w4
   // the same network as SCL:
   #Sollevamento[1].Cin.Rest_ExtEnable := TRUE OR (#AreaInterface.Man AND NOT #CIn.Manager.Sollevamento.Control_ON AND #Sts.OP_CanMoveFreely);
   #Sollevamento[2].Cin.Rest_ExtEnable := TRUE OR (#AreaInterface.Man AND NOT #CIn.Manager.Sollevamento.Control_ON AND #Sts.OP_CanMoveFreely);
   #Sollevamento[3].Cin.Rest_ExtEnable := TRUE OR (#AreaInterface.Man AND NOT #CIn.Manager.Sollevamento.Control_ON AND #Sts.OP_CanMoveFreely);
   #Sollevamento[1].Cin.Work_ExtEnable := #COut.Centraggio.Rest OR (#AreaInterface.Man AND NOT #CIn.Manager.Sollevamento.Control_ON AND #Sts.OP_CanMoveFreely);
   #Sollevamento[2].Cin.Work_ExtEnable := #COut.Centraggio.Rest OR (#AreaInterface.Man AND NOT #CIn.Manager.Sollevamento.Control_ON AND #Sts.OP_CanMoveFreely);
   #Sollevamento[3].Cin.Work_ExtEnable := #COut.Centraggio.Rest OR (#AreaInterface.Man AND NOT #CIn.Manager.Sollevamento.Control_ON AND #Sts.OP_CanMoveFreely);
   #Centraggio[1].Cin.Rest_ExtEnable := TRUE OR (#AreaInterface.Man AND NOT #CIn.Manager.Centraggio.Control_ON AND #Sts.OP_CanMoveFreely);
   #Centraggio[2].Cin.Rest_ExtEnable := TRUE OR (#AreaInterface.Man AND NOT #CIn.Manager.Centraggio.Control_ON AND #Sts.OP_CanMoveFreely);
   #Centraggio[3].Cin.Rest_ExtEnable := TRUE OR (#AreaInterface.Man AND NOT #CIn.Manager.Centraggio.Control_ON AND #Sts.OP_CanMoveFreely);
   #Centraggio[1].Cin.Work_ExtEnable := #COut.Sollevamento.Work OR (#AreaInterface.Man AND NOT #CIn.Manager.Centraggio.Control_ON AND #Sts.OP_CanMoveFreely);
   #Centraggio[2].Cin.Work_ExtEnable := #COut.Sollevamento.Work OR (#AreaInterface.Man AND NOT #CIn.Manager.Centraggio.Control_ON AND #Sts.OP_CanMoveFreely);
   #Centraggio[3].Cin.Work_ExtEnable := #COut.Sollevamento.Work OR (#AreaInterface.Man AND NOT #CIn.Manager.Centraggio.Control_ON AND #Sts.OP_CanMoveFreely);
END_REGION

REGION Network 25: <<< CENTRATORE 1 TESTA >>>
END_REGION

REGION Network 26 (SCL): Centraggio - Finestra di lavoro - Enable/Disable
   // Disattivazione Centratore lato Testa in funzione della posizione del Carro Pareggiatore Testa
   // 

   IF #CIn.CarroPareggTesta.Ax.Homed THEN

       IF #CIn.CarroPareggTesta.Ax.ActualPosition >= "PrjConfig_A03".A0302.Centratori.WorkWindows.Testa.Min AND
           #CIn.CarroPareggTesta.Ax.ActualPosition < "PrjConfig_A03".A0302.Centratori.WorkWindows.Testa.Max THEN
           #Sollevamento[1].Cin.Manager.Rest := TRUE;
           #Centraggio[1].Cin.Manager.Rest := TRUE;
           #HMI.Selection.Sollevamento[1] := FALSE;
           #HMI.Selection.Centraggio[1] := FALSE;
       ELSE
           #HMI.Selection.Sollevamento[1] := TRUE;
           #HMI.Selection.Centraggio[1] := TRUE;
       END_IF;

   ELSE
       #Sollevamento[1].Cin.Manager.Rest := TRUE;
       #Centraggio[1].Cin.Manager.Rest := TRUE;
       #HMI.Selection.Sollevamento[1] := FALSE;
       #HMI.Selection.Centraggio[1] := FALSE;

   END_IF;
END_REGION

REGION Network 27: Centraggio - Valve Machine
   RUNG wire#powerrail
      #Centraggio[1](AreaInterface := #AreaInterface, ZSI := #ZSI, DSI := #DSI, DataIn :=, Cin :=, Config := #Config.Centraggio[1], Alarm := #Alarm.Centraggio[1], Warning := #Warning.Centratore[1], MachineInterface =>, COut =>, DataOut =>)
   END_RUNG
   // the same network as SCL:
   #Centraggio[1](AreaInterface := #AreaInterface,   // "ValveMachine_FB"
                  ZSI := #ZSI,
                  DSI := #DSI,
                  Config := #Config.Centraggio[1],
                  Alarm := #Alarm.Centraggio[1],
                  Warning := #Warning.Centratore[1]);
END_REGION

REGION Network 28: Sollevamento - Valve Machine
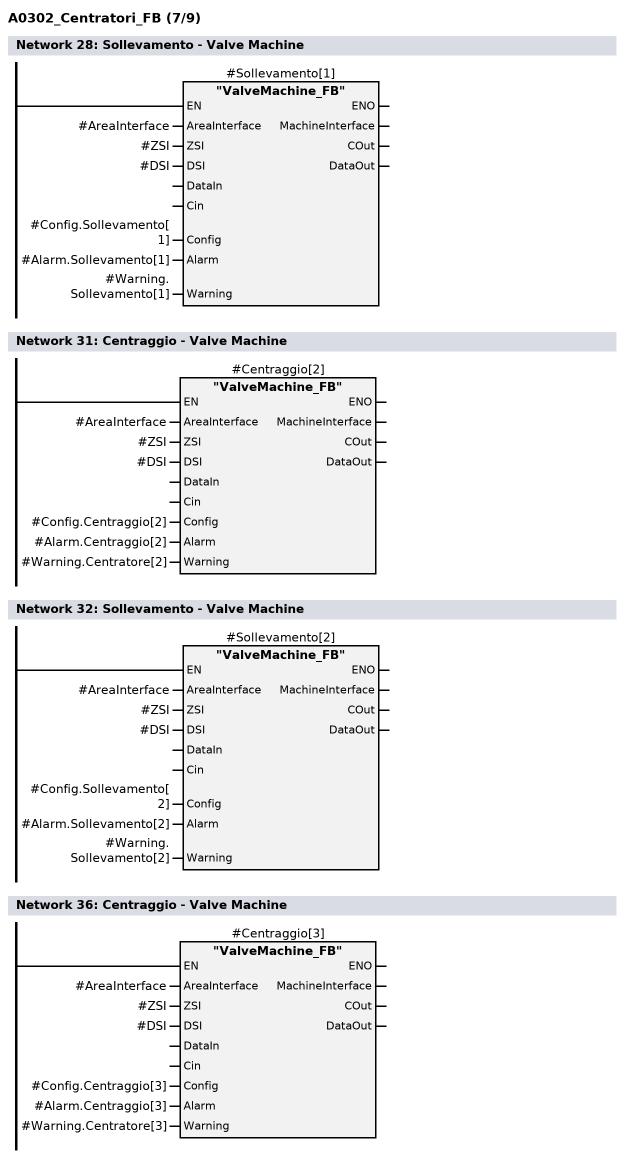
   RUNG wire#powerrail
      #Sollevamento[1](AreaInterface := #AreaInterface, ZSI := #ZSI, DSI := #DSI, DataIn :=, Cin :=, Config := #Config.Sollevamento[1], Alarm := #Alarm.Sollevamento[1], Warning := #Warning.Sollevamento[1], MachineInterface =>, COut =>, DataOut =>)
   END_RUNG
   // the same network as SCL:
   #Sollevamento[1](AreaInterface := #AreaInterface,   // "ValveMachine_FB"
                    ZSI := #ZSI,
                    DSI := #DSI,
                    Config := #Config.Sollevamento[1],
                    Alarm := #Alarm.Sollevamento[1],
                    Warning := #Warning.Sollevamento[1]);
END_REGION

REGION Network 30: <<< CENTRATORE 2 CENTRALE >>>
END_REGION

REGION Network 31: Centraggio - Valve Machine
   RUNG wire#powerrail
      #Centraggio[2](AreaInterface := #AreaInterface, ZSI := #ZSI, DSI := #DSI, DataIn :=, Cin :=, Config := #Config.Centraggio[2], Alarm := #Alarm.Centraggio[2], Warning := #Warning.Centratore[2], MachineInterface =>, COut =>, DataOut =>)
   END_RUNG
   // the same network as SCL:
   #Centraggio[2](AreaInterface := #AreaInterface,   // "ValveMachine_FB"
                  ZSI := #ZSI,
                  DSI := #DSI,
                  Config := #Config.Centraggio[2],
                  Alarm := #Alarm.Centraggio[2],
                  Warning := #Warning.Centratore[2]);
END_REGION

REGION Network 32: Sollevamento - Valve Machine
   RUNG wire#powerrail
      #Sollevamento[2](AreaInterface := #AreaInterface, ZSI := #ZSI, DSI := #DSI, DataIn :=, Cin :=, Config := #Config.Sollevamento[2], Alarm := #Alarm.Sollevamento[2], Warning := #Warning.Sollevamento[2], MachineInterface =>, COut =>, DataOut =>)
   END_RUNG
   // the same network as SCL:
   #Sollevamento[2](AreaInterface := #AreaInterface,   // "ValveMachine_FB"
                    ZSI := #ZSI,
                    DSI := #DSI,
                    Config := #Config.Sollevamento[2],
                    Alarm := #Alarm.Sollevamento[2],
                    Warning := #Warning.Sollevamento[2]);
END_REGION

REGION Network 34: <<< CENTRATORE 3 CODA >>>
END_REGION

REGION Network 35 (SCL): Centraggio - Finestra di lavoro - Enable/Disable
   // Disattivazione Centratore lato Coda in funzione della posizione del Carro Pareggiatore Coda
   // 

   IF #CIn.CarroPareggCoda.Ax.Homed THEN

       IF #CIn.CarroPareggCoda.Ax.ActualPosition >= "PrjConfig_A03".A0302.Centratori.WorkWindows.Coda.Min AND
           #CIn.CarroPareggCoda.Ax.ActualPosition < "PrjConfig_A03".A0302.Centratori.WorkWindows.Coda.Max THEN

           #Sollevamento[3].Cin.Manager.Rest := TRUE;
           #Centraggio[3].Cin.Manager.Rest := TRUE;
           #HMI.Selection.Sollevamento[3] := FALSE;
           #HMI.Selection.Centraggio[3] := FALSE;
       ELSE
           #HMI.Selection.Sollevamento[3] := TRUE;
           #HMI.Selection.Centraggio[3] := TRUE;
       END_IF;

   ELSE
       #Sollevamento[3].Cin.Manager.Rest := TRUE;
       #Centraggio[3].Cin.Manager.Rest := TRUE;
       #HMI.Selection.Sollevamento[3] := FALSE;
       #HMI.Selection.Centraggio[3] := FALSE;

   END_IF;
END_REGION

REGION Network 36: Centraggio - Valve Machine
   RUNG wire#powerrail
      #Centraggio[3](AreaInterface := #AreaInterface, ZSI := #ZSI, DSI := #DSI, DataIn :=, Cin :=, Config := #Config.Centraggio[3], Alarm := #Alarm.Centraggio[3], Warning := #Warning.Centratore[3], MachineInterface =>, COut =>, DataOut =>)
   END_RUNG
   // the same network as SCL:
   #Centraggio[3](AreaInterface := #AreaInterface,   // "ValveMachine_FB"
                  ZSI := #ZSI,
                  DSI := #DSI,
                  Config := #Config.Centraggio[3],
                  Alarm := #Alarm.Centraggio[3],
                  Warning := #Warning.Centratore[3]);
END_REGION

REGION Network 37: Sollevamento - Valve Machine
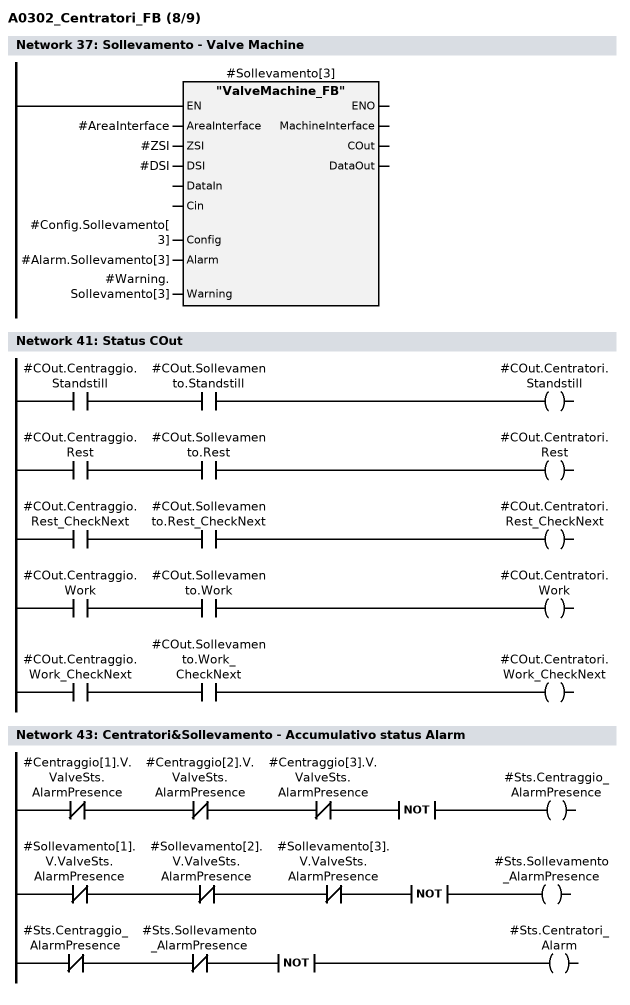
   RUNG wire#powerrail
      #Sollevamento[3](AreaInterface := #AreaInterface, ZSI := #ZSI, DSI := #DSI, DataIn :=, Cin :=, Config := #Config.Sollevamento[3], Alarm := #Alarm.Sollevamento[3], Warning := #Warning.Sollevamento[3], MachineInterface =>, COut =>, DataOut =>)
   END_RUNG
   // the same network as SCL:
   #Sollevamento[3](AreaInterface := #AreaInterface,   // "ValveMachine_FB"
                    ZSI := #ZSI,
                    DSI := #DSI,
                    Config := #Config.Sollevamento[3],
                    Alarm := #Alarm.Sollevamento[3],
                    Warning := #Warning.Sollevamento[3]);
END_REGION

REGION Network 39 (SCL): Centraggio + Sollevamento - COut Centratori
   // Controllo Stato Standstill di tutti i Centraggi
   IF #HMI.Selection.Centraggio[1] AND #HMI.Selection.Centraggio[2] AND #HMI.Selection.Centraggio[3] AND
       #Centraggio[1].Sts.Standstill AND
       #Centraggio[2].Sts.Standstill AND
       #Centraggio[3].Sts.Standstill THEN
       #COut.Centraggio.Standstill := 1;

   ELSIF NOT #HMI.Selection.Centraggio[1] AND #HMI.Selection.Centraggio[2] AND #HMI.Selection.Centraggio[3] AND
       #Centraggio[2].Sts.Standstill AND
       #Centraggio[3].Sts.Standstill THEN
       #COut.Centraggio.Standstill := 1;

   ELSIF #HMI.Selection.Centraggio[1] AND #HMI.Selection.Centraggio[2] AND NOT #HMI.Selection.Centraggio[3] AND
       #Centraggio[1].Sts.Standstill AND
       #Centraggio[2].Sts.Standstill THEN
       #COut.Centraggio.Standstill := 1;

   ELSIF NOT #HMI.Selection.Centraggio[1] AND #HMI.Selection.Centraggio[2] AND NOT #HMI.Selection.Centraggio[3] AND
       #Centraggio[2].Sts.Standstill THEN
       #COut.Centraggio.Standstill := 1;

   ELSE
       #COut.Centraggio.Standstill := 0;
   END_IF;

   // Controllo Stato Standstill di tutti i Sollevamenti

   IF #HMI.Selection.Sollevamento[1] AND #HMI.Selection.Sollevamento[2] AND #HMI.Selection.Sollevamento[3] AND
       #Sollevamento[1].Sts.Standstill AND
       #Sollevamento[2].Sts.Standstill AND
       #Sollevamento[3].Sts.Standstill THEN
       #COut.Sollevamento.Standstill := 1;

   ELSIF NOT #HMI.Selection.Sollevamento[1] AND #HMI.Selection.Sollevamento[2] AND #HMI.Selection.Sollevamento[3] AND
       #Sollevamento[2].Sts.Standstill AND
       #Sollevamento[3].Sts.Standstill THEN
       #COut.Sollevamento.Standstill := 1;

   ELSIF #HMI.Selection.Sollevamento[1] AND #HMI.Selection.Sollevamento[2] AND NOT #HMI.Selection.Sollevamento[3] AND
       #Sollevamento[1].Sts.Standstill AND
       #Sollevamento[2].Sts.Standstill THEN
       #COut.Sollevamento.Standstill := 1;

   ELSIF NOT #HMI.Selection.Sollevamento[1] AND #HMI.Selection.Sollevamento[2] AND NOT #HMI.Selection.Sollevamento[3] AND
       #Sollevamento[2].Sts.Standstill THEN
       #COut.Sollevamento.Standstill := 1;

   ELSE
       #COut.Sollevamento.Standstill := 0;
   END_IF;

   // Controllo uscita COut AT_REST in base allo stato di tutti i Centraggio
   IF #HMI.Selection.Centraggio[1] AND #HMI.Selection.Centraggio[2] AND #HMI.Selection.Centraggio[3] AND
       #Centraggio[1].COut.Rest OR #TON_Anticipi.Rest.Centraggio[1].Q AND
       #Centraggio[2].COut.Rest OR #TON_Anticipi.Rest.Centraggio[2].Q AND
       #Centraggio[3].COut.Rest OR #TON_Anticipi.Rest.Centraggio[3].Q THEN
       #COut.Centraggio.Rest := 1;

   ELSIF NOT #HMI.Selection.Centraggio[1] AND #HMI.Selection.Centraggio[2] AND #HMI.Selection.Centraggio[3] AND
       #Centraggio[2].COut.Rest OR #TON_Anticipi.Rest.Centraggio[2].Q AND
       #Centraggio[3].COut.Rest OR #TON_Anticipi.Rest.Centraggio[3].Q THEN
   #COut.Centraggio.Rest := 1;

   ELSIF #HMI.Selection.Centraggio[1] AND #HMI.Selection.Centraggio[2] AND NOT #HMI.Selection.Centraggio[3] AND
       #Centraggio[1].COut.Rest OR #TON_Anticipi.Rest.Centraggio[1].Q AND
       #Centraggio[2].COut.Rest OR #TON_Anticipi.Rest.Centraggio[2].Q THEN
       #COut.Centraggio.Rest := 1;

   ELSIF NOT #HMI.Selection.Centraggio[1] AND #HMI.Selection.Centraggio[2] AND NOT #HMI.Selection.Centraggio[3] AND
       #Centraggio[2].COut.Rest OR #TON_Anticipi.Rest.Centraggio[2].Q THEN
   #COut.Centraggio.Rest := 1;

   ELSE
   #COut.Centraggio.Rest := 0;
   END_IF;

   // Controllo uscita COut AT_REST in base allo stato di tutti i Sollevamenti
   IF #HMI.Selection.Sollevamento[1] AND #HMI.Selection.Sollevamento[2] AND #HMI.Selection.Sollevamento[3] AND
       #Sollevamento[1].COut.Rest OR #TON_Anticipi.Rest.Sollevamento[1].Q AND
       #Sollevamento[2].COut.Rest OR #TON_Anticipi.Rest.Sollevamento[2].Q AND
       #Sollevamento[3].COut.Rest OR #TON_Anticipi.Rest.Sollevamento[3].Q THEN
       #COut.Sollevamento.Rest := 1;

   ELSIF NOT #HMI.Selection.Sollevamento[1] AND #HMI.Selection.Sollevamento[2] AND #HMI.Selection.Sollevamento[3] AND
       #Sollevamento[2].COut.Rest OR #TON_Anticipi.Rest.Sollevamento[2].Q AND
       #Sollevamento[3].COut.Rest OR #TON_Anticipi.Rest.Sollevamento[3].Q THEN
       #COut.Sollevamento.Rest := 1;

   ELSIF #HMI.Selection.Sollevamento[1] AND #HMI.Selection.Sollevamento[2] AND NOT #HMI.Selection.Sollevamento[3] AND
       #Sollevamento[1].COut.Rest OR #TON_Anticipi.Rest.Sollevamento[1].Q AND
       #Sollevamento[2].COut.Rest OR #TON_Anticipi.Rest.Sollevamento[2].Q THEN
       #COut.Sollevamento.Rest := 1;

   ELSIF NOT #HMI.Selection.Sollevamento[1] AND #HMI.Selection.Sollevamento[2] AND NOT #HMI.Selection.Sollevamento[3] AND
       #Sollevamento[2].COut.Rest OR #TON_Anticipi.Rest.Sollevamento[2].Q THEN
       #COut.Sollevamento.Rest := 1;

   ELSE
       #COut.Sollevamento.Rest := 0;
   END_IF;

   // Controllo uscita COut AT_WORK in base allo stato di tutti i Centraggio
   IF #HMI.Selection.Centraggio[1] AND #HMI.Selection.Centraggio[2] AND #HMI.Selection.Centraggio[3] AND
       #Centraggio[1].COut.Work OR #TON_Anticipi.Rest.Centraggio[1].Q AND
       #Centraggio[2].COut.Work OR #TON_Anticipi.Rest.Centraggio[2].Q AND
       #Centraggio[3].COut.Work OR #TON_Anticipi.Rest.Centraggio[3].Q THEN
       #COut.Centraggio.Work := 1;

   ELSIF NOT #HMI.Selection.Centraggio[1] AND #HMI.Selection.Centraggio[2] AND #HMI.Selection.Centraggio[3] AND
       #Centraggio[2].COut.Work OR #TON_Anticipi.Rest.Centraggio[2].Q AND
       #Centraggio[3].COut.Work OR #TON_Anticipi.Rest.Centraggio[3].Q THEN
       #COut.Centraggio.Work := 1;

   ELSIF #HMI.Selection.Centraggio[1] AND #HMI.Selection.Centraggio[2] AND NOT #HMI.Selection.Centraggio[3] AND
       #Centraggio[1].COut.Work OR #TON_Anticipi.Rest.Centraggio[1].Q AND
       #Centraggio[2].COut.Work OR #TON_Anticipi.Rest.Centraggio[2].Q THEN
       #COut.Centraggio.Work := 1;

   ELSIF NOT #HMI.Selection.Centraggio[1] AND #HMI.Selection.Centraggio[2] AND NOT #HMI.Selection.Centraggio[3] AND
       #Centraggio[2].COut.Work OR #TON_Anticipi.Rest.Centraggio[2].Q THEN
       #COut.Centraggio.Work := 1;

   ELSE
       #COut.Centraggio.Work := 0;
   END_IF;

   // Controllo uscita COut AT_WORK in base allo stato di tutti i Sollevamenti
   IF #HMI.Selection.Sollevamento[1] AND #HMI.Selection.Sollevamento[2] AND #HMI.Selection.Sollevamento[3] AND
       #Sollevamento[1].COut.Work OR #TON_Anticipi.Work.Sollevamento[1].Q AND
       #Sollevamento[2].COut.Work OR #TON_Anticipi.Work.Sollevamento[2].Q AND
       #Sollevamento[3].COut.Work OR #TON_Anticipi.Work.Sollevamento[3].Q THEN
       #COut.Sollevamento.Work := 1;

   ELSIF NOT #HMI.Selection.Sollevamento[1] AND #HMI.Selection.Sollevamento[2] AND #HMI.Selection.Sollevamento[3] AND
       #Sollevamento[2].COut.Work OR #TON_Anticipi.Work.Sollevamento[2].Q AND
       #Sollevamento[3].COut.Work OR #TON_Anticipi.Work.Sollevamento[3].Q THEN
       #COut.Sollevamento.Work := 1;

   ELSIF #HMI.Selection.Sollevamento[1] AND #HMI.Selection.Sollevamento[2] AND NOT #HMI.Selection.Sollevamento[3] AND
       #Sollevamento[1].COut.Work OR #TON_Anticipi.Work.Sollevamento[1].Q AND
       #Sollevamento[2].COut.Work OR #TON_Anticipi.Work.Sollevamento[2].Q THEN
       #COut.Sollevamento.Work := 1;

   ELSIF NOT #HMI.Selection.Sollevamento[1] AND #HMI.Selection.Sollevamento[2] AND NOT #HMI.Selection.Sollevamento[3] AND
       #Sollevamento[2].COut.Work OR #TON_Anticipi.Work.Sollevamento[2].Q THEN
       #COut.Sollevamento.Work := 1;

   ELSE
       #COut.Sollevamento.Work := 0;
   END_IF;
END_REGION

REGION Network 41: Status COut
   RUNG wire#powerrail
      Contact( #COut.Centraggio.Standstill )
      Contact( #COut.Sollevamento.Standstill )
      Coil( #COut.Centratori.Standstill )
   END_RUNG
   RUNG wire#powerrail
      Contact( #COut.Centraggio.Rest )
      Contact( #COut.Sollevamento.Rest )
      Coil( #COut.Centratori.Rest )
   END_RUNG
   RUNG wire#powerrail
      Contact( #COut.Centraggio.Rest_CheckNext )
      Contact( #COut.Sollevamento.Rest_CheckNext )
      Coil( #COut.Centratori.Rest_CheckNext )
   END_RUNG
   RUNG wire#powerrail
      Contact( #COut.Centraggio.Work )
      Contact( #COut.Sollevamento.Work )
      Coil( #COut.Centratori.Work )
   END_RUNG
   RUNG wire#powerrail
      Contact( #COut.Centraggio.Work_CheckNext )
      Contact( #COut.Sollevamento.Work_CheckNext )
      Coil( #COut.Centratori.Work_CheckNext )
   END_RUNG
   // the same network as SCL:
   #COut.Centratori.Standstill := #COut.Centraggio.Standstill AND #COut.Sollevamento.Standstill;
   #COut.Centratori.Rest := #COut.Centraggio.Rest AND #COut.Sollevamento.Rest;
   #COut.Centratori.Rest_CheckNext := #COut.Centraggio.Rest_CheckNext AND #COut.Sollevamento.Rest_CheckNext;
   #COut.Centratori.Work := #COut.Centraggio.Work AND #COut.Sollevamento.Work;
   #COut.Centratori.Work_CheckNext := #COut.Centraggio.Work_CheckNext AND #COut.Sollevamento.Work_CheckNext;
END_REGION

REGION Network 43: Centratori&Sollevamento - Accumulativo status Alarm
   RUNG wire#powerrail
      I_Contact( #Centraggio[1].V.ValveSts.AlarmPresence )
      I_Contact( #Centraggio[2].V.ValveSts.AlarmPresence )
      I_Contact( #Centraggio[3].V.ValveSts.AlarmPresence )
      Not()
      Coil( #Sts.Centraggio_AlarmPresence )
   END_RUNG
   RUNG wire#powerrail
      I_Contact( #Sollevamento[1].V.ValveSts.AlarmPresence )
      I_Contact( #Sollevamento[2].V.ValveSts.AlarmPresence )
      I_Contact( #Sollevamento[3].V.ValveSts.AlarmPresence )
      Not()
      Coil( #Sts.Sollevamento_AlarmPresence )
   END_RUNG
   RUNG wire#powerrail
      I_Contact( #Sts.Centraggio_AlarmPresence )
      I_Contact( #Sts.Sollevamento_AlarmPresence )
      Not()
      Coil( #Sts.Centratori_Alarm )
   END_RUNG
   // the same network as SCL:
   #Sts.Centraggio_AlarmPresence := NOT (NOT #Centraggio[1].V.ValveSts.AlarmPresence AND NOT #Centraggio[2].V.ValveSts.AlarmPresence AND NOT #Centraggio[3].V.ValveSts.AlarmPresence);
   #Sts.Sollevamento_AlarmPresence := NOT (NOT #Sollevamento[1].V.ValveSts.AlarmPresence AND NOT #Sollevamento[2].V.ValveSts.AlarmPresence AND NOT #Sollevamento[3].V.ValveSts.AlarmPresence);
   #Sts.Centratori_Alarm := NOT (NOT #Sts.Centraggio_AlarmPresence AND NOT #Sts.Sollevamento_AlarmPresence);
END_REGION

REGION Network 44 (SCL): HMI STATUS - Postazione
   // Area dati appoggio per HMI
   // CENTRATORI
   #HMI.Centraggio_Sts.Standstill := #COut.Centraggio.Standstill;
   #HMI.Centraggio_Sts.Rest := #COut.Centraggio.Rest;
   #HMI.Centraggio_Sts.Work := #COut.Centraggio.Work;
   #HMI.Centraggio_Sts.AlarmPresence := #Sts.Centraggio_AlarmPresence;

   // SOLLEVAMENTO
   #HMI.Sollevamento_Sts.Standstill := #COut.Sollevamento.Standstill;
   #HMI.Sollevamento_Sts.Rest := #COut.Sollevamento.Rest;
   #HMI.Sollevamento_Sts.Work := #COut.Sollevamento.Work;
   #HMI.Sollevamento_Sts.AlarmPresence := #Sts.Sollevamento_AlarmPresence;

   // STAZIONE CENTRATORI
   #HMI.Centratori_Sts.Standstill := #COut.Centratori.Standstill;
   #HMI.Centratori_Sts.Rest := #COut.Centratori.Rest;
   #HMI.Centratori_Sts.Work := #COut.Centratori.Work;
   #HMI.Centratori_Sts.AlarmPresence := #Sts.Centratori_Alarm;
END_REGION

REGION Network 45: <<< MACHINE STATUS >>>
END_REGION

REGION Network 46: Collect machine to zone interface (internal machines OR)
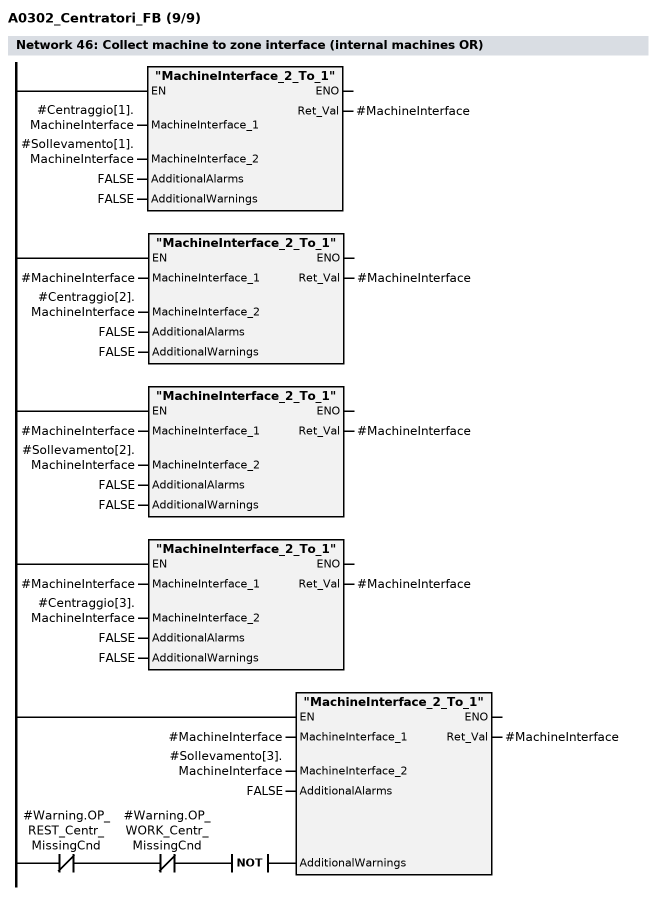
   RUNG wire#powerrail
      "MachineInterface_2_To_1"(MachineInterface_1 := #Centraggio[1].MachineInterface, MachineInterface_2 := #Sollevamento[1].MachineInterface, AdditionalAlarms := FALSE, AdditionalWarnings := FALSE, Ret_Val => #MachineInterface)
   END_RUNG
   RUNG wire#powerrail
      "MachineInterface_2_To_1"(MachineInterface_1 := #MachineInterface, MachineInterface_2 := #Centraggio[2].MachineInterface, AdditionalAlarms := FALSE, AdditionalWarnings := FALSE, Ret_Val => #MachineInterface)
   END_RUNG
   RUNG wire#powerrail
      "MachineInterface_2_To_1"(MachineInterface_1 := #MachineInterface, MachineInterface_2 := #Sollevamento[2].MachineInterface, AdditionalAlarms := FALSE, AdditionalWarnings := FALSE, Ret_Val => #MachineInterface)
   END_RUNG
   RUNG wire#powerrail
      "MachineInterface_2_To_1"(MachineInterface_1 := #MachineInterface, MachineInterface_2 := #Centraggio[3].MachineInterface, AdditionalAlarms := FALSE, AdditionalWarnings := FALSE, Ret_Val => #MachineInterface)
   END_RUNG
   RUNG wire#powerrail
      "MachineInterface_2_To_1"(AdditionalWarnings := wire#w1, MachineInterface_1 := #MachineInterface, MachineInterface_2 := #Sollevamento[3].MachineInterface, AdditionalAlarms := FALSE, Ret_Val => #MachineInterface)
   END_RUNG
   RUNG wire#powerrail
      I_Contact( #Warning.OP_REST_Centr_MissingCnd )
      I_Contact( #Warning.OP_WORK_Centr_MissingCnd )
      Not()
   END_RUNG wire#w1
   // the same network as SCL:
   #MachineInterface := "MachineInterface_2_To_1"(MachineInterface_1 := #Centraggio[1].MachineInterface,
                           MachineInterface_2 := #Sollevamento[1].MachineInterface,
                           AdditionalAlarms := FALSE,
                           AdditionalWarnings := FALSE);
   #MachineInterface := "MachineInterface_2_To_1"(MachineInterface_1 := #MachineInterface,
                           MachineInterface_2 := #Centraggio[2].MachineInterface,
                           AdditionalAlarms := FALSE,
                           AdditionalWarnings := FALSE);
   #MachineInterface := "MachineInterface_2_To_1"(MachineInterface_1 := #MachineInterface,
                           MachineInterface_2 := #Sollevamento[2].MachineInterface,
                           AdditionalAlarms := FALSE,
                           AdditionalWarnings := FALSE);
   #MachineInterface := "MachineInterface_2_To_1"(MachineInterface_1 := #MachineInterface,
                           MachineInterface_2 := #Centraggio[3].MachineInterface,
                           AdditionalAlarms := FALSE,
                           AdditionalWarnings := FALSE);
   #MachineInterface := "MachineInterface_2_To_1"(MachineInterface_1 := #MachineInterface,
                           MachineInterface_2 := #Sollevamento[3].MachineInterface,
                           AdditionalAlarms := FALSE,
                           AdditionalWarnings := NOT (NOT #Warning.OP_REST_Centr_MissingCnd AND NOT #Warning.OP_WORK_Centr_MissingCnd));
END_REGION
END_FUNCTION_BLOCK

FUNCTION "FcP_R_Trig" : Void
{ S7_Optimized_Access := 'TRUE' ; Published := 'FALSE' }
VERSION : 0.1
//Rising edge detection
   VAR_INPUT 
      CLK : Bool;   // Input to detect rising edge
   END_VAR

   VAR_OUTPUT 
      Q : Bool;   // Pulse output
   END_VAR

   VAR_IN_OUT 
      M : Bool;   // Memory bit
   END_VAR


BEGIN
	#Q := #CLK AND NOT #M; // Calculate rising edge
	#M := #CLK; // Copy input to storage bit
END_FUNCTION

FUNCTION "GetEFCErrorCode" : Word
{ S7_Optimized_Access := 'TRUE' ; Published := 'FALSE' }
VERSION : 0.1
   VAR_INPUT 
      EFCStatusWord : "EFC_STATUS_WORD";   // EFC status word
      Prefix : Word;   // Prefix for error code
   END_VAR


BEGIN
	#GetEFCErrorCode := "PrefixCode"(Value := "GetErrorCode"(EFCStatusWord := #EFCStatusWord), "Prefix" := #Prefix); // Return error code with prefix value
	
	
END_FUNCTION

FUNCTION "PrefixCode" : Word
{ S7_Optimized_Access := 'TRUE' ; Published := 'FALSE' }
VERSION : 0.1
   VAR_INPUT 
      Value : Word;   // Error / warning code
      Prefix : Word;   // Prefix for error / warning code
   END_VAR


BEGIN
	#PrefixCode := #Value + #Prefix;
END_FUNCTION

FUNCTION "GetFcPCode" : Word
{ S7_Optimized_Access := 'TRUE' ; Published := 'FALSE' }
VERSION : 0.1
   VAR_INPUT 
      Value : Word;
      Prefix : Word;
      Min : Word;
      Max : Word;
      ValueIsDecimal : Bool;
   END_VAR

   VAR_TEMP 
      wValue : Word;
   END_VAR


BEGIN
	IF (#Value < #Min) OR (#Value > #Max) THEN
	    #GetFcPCode := #Prefix;
	    RETURN;
	ELSE
	    IF (#ValueIsDecimal = TRUE) THEN
	        #wValue := "DecToHexNumber"(Value := #Value);
	    ELSE
	        #wValue := #Value;
	    END_IF;
	    #GetFcPCode := "PrefixCode"(Prefix := #Prefix, Value := #wValue);
	END_IF;
	
	
	
END_FUNCTION

FUNCTION "SwapWord" : Word
{ S7_Optimized_Access := 'TRUE' ; Published := 'FALSE' }
VERSION : 0.1
   VAR_INPUT 
      WordIn : Word;
   END_VAR

   VAR_TEMP 
      wIn : Word;
      arInput : Array[1..2] of Byte;
      wOut : Word;
      arOutput : Array[1..2] of Byte;
   END_VAR


BEGIN
	#wIn := #WordIn;
	
	// Scompongo Word ingresso
	#arInput[1] := WORD_TO_BYTE(IN := #wIn);
	#arInput[2] := WORD_TO_BYTE(IN := SHR(IN := #wIn, N := 8));
	
	// Swap dei Byte
	#arOutput[1] := #arInput[2];
	#arOutput[2] := #arInput[1];
	
	//Compongo la Word di uscita
	#wOut := BYTE_TO_WORD(IN := #arOutput[1]) OR (BYTE_TO_WORD(IN:= SHL(IN := #arOutput[2],N:=8)));
	                       
	#SwapWord := #wOut;
	                       
	                       
END_FUNCTION

DATA_BLOCK "Area03"   // DB40
// stored: InstanceOfName Area, InstanceOfType FB
"Area"
   // VAR_INPUT
   //    Estop : Bool;
   //    DataIn : Struct
   //       SelMan : Bool;
   //       SelAut : Bool;
   //       PbStart : Bool;
   //       PbStop : Bool;
   //       PbStopProgrammed : Bool;
   //       PbAckRst : Bool;
   //    END_STRUCT;
   //    Config : "AreaConfig";
   //    MachinesStatus : "MachineStatus";
   //    ForceStopInPhase : Bool;
   //    ForceStopProgrammed : Bool;
   //    ResetTimersTimeoutStops : Bool;
   // END_VAR
   // VAR_OUTPUT
   //    AreaInterface { ExternalVisible := 'False'; ExternalWritable := 'False'} : "AreaInterface";
   //    DataOut : Struct
   //       horn : Bool;
   //       lampReady : Bool;
   //       lampCycle : Bool;
   //       LampWarningPresence : Bool;
   //       LampAlarmPresence : Bool;
   //    END_STRUCT;
   //    SilencingAlarms : Bool;
   //    HMI_StatusDinamicText : Int;
   // END_VAR
   // VAR
   //    pbStartOneShotAux : Bool;
   //    RstAlrOneShot1 : Bool;
   //    RstAlrOneShot2 : Bool;
   //    CycleStopImmediately : Bool;
   //    CycleStopInPhase : Bool;
   //    CycleStarted : Bool;
   //    CycleStopProgrammed : Bool;
   //    CycleOn : Bool;
   //    ManAuxPe : Bool;
   //    ManAuxNe : Bool;
   //    ManPositiveEdge : Bool;
   //    ManNegativeEdge : Bool;
   //    AutAuxPe : Bool;
   //    AutAuxNe : Bool;
   //    AutPositiveEdge : Bool;
   //    AutNegativeEdge : Bool;
   //    AlarmLAuxPe : Bool;
   //    CycleAuxPe : Bool;
   //    ResetAlarmsCmd : Bool;
   //    tonDelayPbStart { S7_SetPoint := 'True'} : IEC_TIMER;
   //    tonDelayRstAck { S7_SetPoint := 'True'} : IEC_TIMER;
   //    tonTimeOutStopPhase { S7_SetPoint := 'True'} : IEC_TIMER;
   //    tonTimeOutStopProgr { S7_SetPoint := 'True'} : IEC_TIMER;
   //    tonTimeOutResetAlr { S7_SetPoint := 'True'} : IEC_TIMER;
   // END_VAR
BEGIN
END_DATA_BLOCK

DATA_BLOCK "Area03_Msg_Alarms"   // DB106
// stored: InstanceOfName MsgManager, InstanceOfType FB
"MsgManager"
   // VAR_INPUT
   //    Ack : Bool;
   // END_VAR
   // VAR_OUTPUT
   //    MessagePresence : Bool;
   //    NewMessage : Bool;
   //    MessageCount : Int;
   // END_VAR
   // VAR_IN_OUT
   //    Messages : Array[*] of Bool;
   //    MessagesHMI : Array[*] of Word;
   //    MessagesACK : Array[*] of Word;
   // END_VAR
   // VAR
   //    MsgDim : DInt;
   //    HmiMsgDim : DInt;
   //    AckMsgDim : DInt;
   //    MsgCount : Int;
   //    Status : Int;
   //    IndexBuild : Int;
   //    IndexCompare : Int;
   //    LoopStart : Int;
   //    LoopEnd : Int;
   //    HMIIndex : Int;
   //    CompareWord : Word;
   //    "A" : Word;
   //    MvBlkVar_ErrorID : Int;
   // END_VAR
BEGIN
END_DATA_BLOCK

DATA_BLOCK "Area03_Msg_Warnings"   // DB24
// stored: InstanceOfName MsgManager, InstanceOfType FB
"MsgManager"
   // VAR_INPUT
   //    Ack : Bool;
   // END_VAR
   // VAR_OUTPUT
   //    MessagePresence : Bool;
   //    NewMessage : Bool;
   //    MessageCount : Int;
   // END_VAR
   // VAR_IN_OUT
   //    Messages : Array[*] of Bool;
   //    MessagesHMI : Array[*] of Word;
   //    MessagesACK : Array[*] of Word;
   // END_VAR
   // VAR
   //    MsgDim : DInt;
   //    HmiMsgDim : DInt;
   //    AckMsgDim : DInt;
   //    MsgCount : Int;
   //    Status : Int;
   //    IndexBuild : Int;
   //    IndexCompare : Int;
   //    LoopStart : Int;
   //    LoopEnd : Int;
   //    HMIIndex : Int;
   //    CompareWord : Word;
   //    "A" : Word;
   //    MvBlkVar_ErrorID : Int;
   // END_VAR
BEGIN
END_DATA_BLOCK

DATA_BLOCK "A03_HMI_IDB"   // DB72
AUTHOR : Piemme
FAMILY : System
// stored: InstanceOfName HMI_A03_FB, InstanceOfType FB
"HMI_A03_FB"
BEGIN
END_DATA_BLOCK

DATA_BLOCK "A03_0102TrkManager"   // DB188
// stored: InstanceOfName A03_0102TrkManager_FB, InstanceOfType FB
"A03_0102TrkManager_FB"
   // VAR_INPUT
   //    AreaInterface : "AreaInterface";
   //    SuperUserLogged : Bool;
   // END_VAR
   // VAR
   //    HMI : Struct
   //       A0301_P : Struct
   //          Move : Array[1..11] of "TrkMng_Move";
   //       END_STRUCT;
   //       A0301_B : Struct
   //          Move : Array[1..12] of "TrkMng_Move";
   //       END_STRUCT;
   //       A0302_ENTRY : Struct
   //          Move : Array[1..7] of "TrkMng_Move";
   //       END_STRUCT;
   //       A0302_EXIT : Struct
   //          Move : Array[1..18] of "TrkMng_Move";
   //       END_STRUCT;
   //    END_STRUCT;
   //    Sts : Struct
   //       MoveA0301_P : Struct
   //          SelectionOn : Bool;
   //          SelectionNo : Int;
   //       END_STRUCT;
   //       MoveA0301_B : Struct
   //          SelectionOn : Bool;
   //          SelectionNo : Int;
   //       END_STRUCT;
   //       MoveA0302_ENTRY : Struct
   //          SelectionOn : Bool;
   //          SelectionNo : Int;
   //       END_STRUCT;
   //       MoveA0302_EXIT : Struct
   //          SelectionOn : Bool;
   //          SelectionNo : Int;
   //       END_STRUCT;
   //    END_STRUCT;
   //    A0301B_TON_Delete_Buttons : IEC_TIMER;
   //    A0301P_TON_Delete_Buttons : IEC_TIMER;
   //    A0302_ENTRY_TON_Delete_Buttons : IEC_TIMER;
   //    A0302_EXIT_TON_Delete_Buttons : IEC_TIMER;
   // END_VAR
BEGIN
END_DATA_BLOCK

DATA_BLOCK "A0301_Manager"   // DB23
// stored: InstanceOfName A0301_Manager_FB, InstanceOfType FB
"A0301_Manager_FB"
BEGIN
END_DATA_BLOCK

DATA_BLOCK "A0301_Trasporto"   // DB75
// stored: InstanceOfName A0301_Trasporto_FB, InstanceOfType FB
"A0301_Trasporto_FB"
BEGIN
END_DATA_BLOCK

DATA_BLOCK "A0301_Fermi_P1"   // DB51
// stored: InstanceOfName A0301_Fermi_P1_FB, InstanceOfType FB
"A0301_Fermi_P1_FB"
BEGIN
   AreaInterface.EStop := FALSE;
   AreaInterface.Man := TRUE;
   AreaInterface.Aut := FALSE;
   AreaInterface.Cycle := FALSE;
   AreaInterface.StopInPhase := FALSE;
   AreaInterface.StopProgrammed := FALSE;
   AreaInterface.RstAlarms := FALSE;
   AreaInterface.ManOneShot := FALSE;
   AreaInterface.AutOneShot := FALSE;
   AreaInterface.CycleOneShot := FALSE;
   AreaInterface.CheckAutReady := FALSE;
   ZSI.Door_NormalStop := FALSE;
   ZSI.Door_SafeStop := FALSE;
   ZSI.Door_Opened := FALSE;
   ZSI.Door_EntryEnable := FALSE;
   DSI.SafeStop := FALSE;
   DSI.PowerEnable := TRUE;
   DSI.DevicesInSafeState := FALSE;
   CIn.Manager_Fermi.EnableStopDoorOpeningReq := FALSE;
   CIn.Manager_Fermi.EnableStopInPhase := FALSE;
   CIn.Manager_Fermi.EnableStopProgrammed := FALSE;
   CIn.Manager_Fermi.Control_ON := FALSE;
   CIn.Manager_Fermi.Rest := FALSE;
   CIn.Manager_Fermi.Work := FALSE;
   CIn.Trasporto.Infeed_ReqON := FALSE;
   CIn.Trasporto.CtrlSafe := FALSE;
   CIn.Trasporto.Standstill := TRUE;
   CIn.Trasporto.Bwd_CheckNext := FALSE;
   CIn.Trasporto.Fwd_CheckNext := FALSE;
   CIn.Trasporto.Bwd_VelZero := FALSE;
   CIn.Trasporto.Bwd_Running := FALSE;
   CIn.Trasporto.Fwd_VelZero := FALSE;
   CIn.Trasporto.Fwd_Running := FALSE;
   CIn.Trasporto.ActualVelocity := 0.0;
   CIn.Trasporto.TargetVelocity := 0.0;
   CIn.Trasporto.MaxVelocity := 39597.8;
   Config.Fermi[1..6].DelayPressureRunningTimeout := T#3S;
   Config.Fermi[1..6].DelayMissingCondition := T#3S;
   Config.Fermi[1..6].Rest_LsQty := 1;
   Config.Fermi[1..6].Work_LsQty := 0;
   Config.Fermi[1..6].Rest_RetainAut := FALSE;
   Config.Fermi[1..6].Work_RetainAut := FALSE;
   Config.Fermi[1..6].V.RestLimSwitchExist := TRUE;
   Config.Fermi[1..6].V.WorkLimSwitchExist := FALSE;
   Config.Fermi[1..6].V.CheckOilInPressure := FALSE;
   Config.Fermi[1..6].V.CutRestWhenIsAtRest := TRUE;
   Config.Fermi[1..6].V.CutWorkWhenIsAtWork := TRUE;
   Config.Fermi[1..6].V.RestTime := T#2S;
   Config.Fermi[1..6].V.WorkTime := T#2S;
   Config.Fermi[1..6].V.RestTimeOut := T#4S;
   Config.Fermi[1..6].V.WorkTimeOut := T#4S;
   Config.Pareggiatore.DelayPressureRunningTimeout := T#3S;
   Config.Pareggiatore.DelayMissingCondition := T#3S;
   Config.Pareggiatore.Rest_LsQty := 1;
   Config.Pareggiatore.Work_LsQty := 1;
   Config.Pareggiatore.Rest_RetainAut := FALSE;
   Config.Pareggiatore.Work_RetainAut := FALSE;
   Config.Pareggiatore.V.RestLimSwitchExist := TRUE;
   Config.Pareggiatore.V.WorkLimSwitchExist := TRUE;
   Config.Pareggiatore.V.CheckOilInPressure := FALSE;
   Config.Pareggiatore.V.CutRestWhenIsAtRest := TRUE;
   Config.Pareggiatore.V.CutWorkWhenIsAtWork := TRUE;
   Config.Pareggiatore.V.RestTime := T#1S;
   Config.Pareggiatore.V.WorkTime := T#1S;
   Config.Pareggiatore.V.RestTimeOut := T#1H;
   Config.Pareggiatore.V.WorkTimeOut := T#1H;
   MachineInterface.AutReady := FALSE;
   MachineInterface.Aborting := FALSE;
   MachineInterface.AckStopInPhase := FALSE;
   MachineInterface.AckStopProgrammed := FALSE;
   MachineInterface.MotionsStandStill := TRUE;
   MachineInterface.AlarmsPresence := FALSE;
   MachineInterface.WarningPresence := FALSE;
   COut.Fermi.CtrlSafe := FALSE;
   COut.Fermi.Standstill := TRUE;
   COut.Fermi.ReqOilPressure := FALSE;
   COut.Fermi.Rest_CheckNext := FALSE;
   COut.Fermi.Work_CheckNext := FALSE;
   COut.Fermi.Rest := FALSE;
   COut.Fermi.Work := FALSE;
   COut.Pareggiatore.CtrlSafe := FALSE;
   COut.Pareggiatore.Standstill := TRUE;
   COut.Pareggiatore.ReqOilPressure := FALSE;
   COut.Pareggiatore.Rest_CheckNext := FALSE;
   COut.Pareggiatore.Work_CheckNext := FALSE;
   COut.Pareggiatore.Rest := FALSE;
   COut.Pareggiatore.Work := FALSE;
   Alarm.Fermi[1..6].TimeOutRest := FALSE;
   Alarm.Fermi[1..6].TimeOutWork := FALSE;
   Alarm.Fermi[1..6].LimitSwitches := FALSE;
   Alarm.Pareggiatore.TimeOutRest := FALSE;
   Alarm.Pareggiatore.TimeOutWork := FALSE;
   Alarm.Pareggiatore.LimitSwitches := FALSE;
   Warning.Fermi[1..6].NotAutReady := FALSE;
   Warning.Fermi[1..6].PressureRunning_Timeout := FALSE;
   Warning.Fermi[1..6].Rest_MissingExtEnable := FALSE;
   Warning.Fermi[1..6].Work_MissingExtEnable := FALSE;
   Warning.Fermi[1].Missing_Rest_Ls_ON[1..8] := FALSE;
   Warning.Fermi[2].Missing_Rest_Ls_ON[1..8] := FALSE;
   Warning.Fermi[3].Missing_Rest_Ls_ON[1..8] := FALSE;
   Warning.Fermi[4].Missing_Rest_Ls_ON[1..8] := FALSE;
   Warning.Fermi[5].Missing_Rest_Ls_ON[1..8] := FALSE;
   Warning.Fermi[6].Missing_Rest_Ls_ON[1..8] := FALSE;
   Warning.Fermi[1].Missing_Work_Ls_ON[1..8] := FALSE;
   Warning.Fermi[2].Missing_Work_Ls_ON[1..8] := FALSE;
   Warning.Fermi[3].Missing_Work_Ls_ON[1..8] := FALSE;
   Warning.Fermi[4].Missing_Work_Ls_ON[1..8] := FALSE;
   Warning.Fermi[5].Missing_Work_Ls_ON[1..8] := FALSE;
   Warning.Fermi[6].Missing_Work_Ls_ON[1..8] := FALSE;
   Warning.Pareggiatore.NotAutReady := FALSE;
   Warning.Pareggiatore.PressureRunning_Timeout := FALSE;
   Warning.Pareggiatore.Rest_MissingExtEnable := FALSE;
   Warning.Pareggiatore.Work_MissingExtEnable := FALSE;
   Warning.Pareggiatore.Missing_Rest_Ls_ON[1..8] := FALSE;
   Warning.Pareggiatore.Missing_Work_Ls_ON[1..8] := FALSE;
   HMI.Selection[1..6] := TRUE;
   HMI.FermiSts.Standstill := TRUE;
   HMI.FermiSts.Rest := FALSE;
   HMI.FermiSts.Work := FALSE;
   HMI.FermiSts.AlarmPresence := FALSE;
   HMI.PareggiatoreSts.Standstill := TRUE;
   HMI.PareggiatoreSts.Rest := FALSE;
   HMI.PareggiatoreSts.Work := FALSE;
   HMI.PareggiatoreSts.AlarmPresence := FALSE;
   Fermi[1..6].AreaInterface.EStop := FALSE;
   Fermi[1..6].AreaInterface.Man := TRUE;
   Fermi[1..6].AreaInterface.Aut := FALSE;
   Fermi[1..6].AreaInterface.Cycle := FALSE;
   Fermi[1..6].AreaInterface.StopInPhase := FALSE;
   Fermi[1..6].AreaInterface.StopProgrammed := FALSE;
   Fermi[1..6].AreaInterface.RstAlarms := FALSE;
   Fermi[1..6].AreaInterface.ManOneShot := FALSE;
   Fermi[1..6].AreaInterface.AutOneShot := FALSE;
   Fermi[1..6].AreaInterface.CycleOneShot := FALSE;
   Fermi[1..6].AreaInterface.CheckAutReady := FALSE;
   Fermi[1..6].ZSI.Door_NormalStop := FALSE;
   Fermi[1..6].ZSI.Door_SafeStop := FALSE;
   Fermi[1..6].ZSI.Door_Opened := FALSE;
   Fermi[1..6].ZSI.Door_EntryEnable := FALSE;
   Fermi[1..6].DSI.SafeStop := FALSE;
   Fermi[1..6].DSI.PowerEnable := TRUE;
   Fermi[1..6].DSI.DevicesInSafeState := FALSE;
   Fermi[1..6].DataIn.PB.Rest := FALSE;
   Fermi[1..6].DataIn.PB.Work := FALSE;
   Fermi[1..6].DataIn.PB.StartStop := FALSE;
   Fermi[1].DataIn.Rest_Ls[1] := TRUE;
   Fermi[1].DataIn.Rest_Ls[2..8] := FALSE;
   Fermi[2].DataIn.Rest_Ls[1] := TRUE;
   Fermi[2].DataIn.Rest_Ls[2..8] := FALSE;
   Fermi[3].DataIn.Rest_Ls[1] := TRUE;
   Fermi[3].DataIn.Rest_Ls[2..8] := FALSE;
   Fermi[4].DataIn.Rest_Ls[1] := TRUE;
   Fermi[4].DataIn.Rest_Ls[2..8] := FALSE;
   Fermi[5].DataIn.Rest_Ls[1] := TRUE;
   Fermi[5].DataIn.Rest_Ls[2..8] := FALSE;
   Fermi[6].DataIn.Rest_Ls[1] := TRUE;
   Fermi[6].DataIn.Rest_Ls[2..8] := FALSE;
   Fermi[1].DataIn.Work_Ls[1..8] := FALSE;
   Fermi[2].DataIn.Work_Ls[1..8] := FALSE;
   Fermi[3].DataIn.Work_Ls[1..8] := FALSE;
   Fermi[4].DataIn.Work_Ls[1..8] := FALSE;
   Fermi[5].DataIn.Work_Ls[1..8] := FALSE;
   Fermi[6].DataIn.Work_Ls[1..8] := FALSE;
   Fermi[1..6].Cin.Manager.EnableStopDoorOpeningReq := FALSE;
   Fermi[1..6].Cin.Manager.EnableStopInPhase := FALSE;
   Fermi[1..6].Cin.Manager.EnableStopProgrammed := FALSE;
   Fermi[1..6].Cin.Manager.Control_ON := FALSE;
   Fermi[1..6].Cin.Manager.Rest := FALSE;
   Fermi[1..6].Cin.Manager.Work := FALSE;
   Fermi[1..6].Cin.PressureRunning := FALSE;
   Fermi[1..6].Cin.Rest_ExtEnable := TRUE;
   Fermi[1..6].Cin.Work_ExtEnable := TRUE;
   Fermi[1..6].Cin.ExternalAlarms := FALSE;
   Fermi[1..6].Config.DelayPressureRunningTimeout := T#3S;
   Fermi[1..6].Config.DelayMissingCondition := T#3S;
   Fermi[1..6].Config.Rest_LsQty := 1;
   Fermi[1..6].Config.Work_LsQty := 0;
   Fermi[1..6].Config.Rest_RetainAut := FALSE;
   Fermi[1..6].Config.Work_RetainAut := FALSE;
   Fermi[1..6].Config.V.RestLimSwitchExist := TRUE;
   Fermi[1..6].Config.V.WorkLimSwitchExist := FALSE;
   Fermi[1..6].Config.V.CheckOilInPressure := FALSE;
   Fermi[1..6].Config.V.CutRestWhenIsAtRest := TRUE;
   Fermi[1..6].Config.V.CutWorkWhenIsAtWork := TRUE;
   Fermi[1..6].Config.V.RestTime := T#2S;
   Fermi[1..6].Config.V.WorkTime := T#2S;
   Fermi[1..6].Config.V.RestTimeOut := T#4S;
   Fermi[1..6].Config.V.WorkTimeOut := T#4S;
   Fermi[1..6].MachineInterface.AutReady := FALSE;
   Fermi[1..6].MachineInterface.Aborting := FALSE;
   Fermi[1..6].MachineInterface.AckStopInPhase := FALSE;
   Fermi[1..6].MachineInterface.AckStopProgrammed := FALSE;
   Fermi[1..6].MachineInterface.MotionsStandStill := TRUE;
   Fermi[1..6].MachineInterface.AlarmsPresence := FALSE;
   Fermi[1..6].MachineInterface.WarningPresence := FALSE;
   Fermi[1..6].COut.CtrlSafe := FALSE;
   Fermi[1..6].COut.Standstill := TRUE;
   Fermi[1..6].COut.ReqOilPressure := FALSE;
   Fermi[1..6].COut.Rest_CheckNext := FALSE;
   Fermi[1..6].COut.Work_CheckNext := FALSE;
   Fermi[1..6].COut.Rest := TRUE;
   Fermi[1..6].COut.Work := FALSE;
   Fermi[1..6].DataOut.RestSolenoid := FALSE;
   Fermi[1..6].DataOut.WorkSolenoid := FALSE;
   Fermi[1..6].Sts.Standstill := TRUE;
   Fermi[1..6].Sts.AlarmsPresence := FALSE;
   Fermi[1..6].Sts.WarningsPresence := FALSE;
   Fermi[1..6].Sts.Rest_Cnd := TRUE;
   Fermi[1..6].Sts.Work_Cnd := TRUE;
   Fermi[1..6].Ctrl.StopDueDoorOpeningRequest := FALSE;
   Fermi[1..6].Ctrl.StopInPhase := FALSE;
   Fermi[1..6].Ctrl.StopProgrammed := FALSE;
   Fermi[1..6].Ctrl.StopAborting := FALSE;
   Fermi[1..6].Ctrl.Work := FALSE;
   Fermi[1..6].Ctrl.Rest := FALSE;
   Fermi[1..6].Ctrl.Rest_Man := FALSE;
   Fermi[1..6].Ctrl.Work_Man := FALSE;
   Fermi[1..6].Ctrl.Rest_Aut := FALSE;
   Fermi[1..6].Ctrl.Work_Aut := FALSE;
   Fermi[1..6].V.ValveCtrl.SafeStop := FALSE;
   Fermi[1..6].V.ValveCtrl.Rst := FALSE;
   Fermi[1..6].V.ValveCtrl.MoveRest := FALSE;
   Fermi[1..6].V.ValveCtrl.MoveWork := FALSE;
   Fermi[1..6].V.RestLimitSwitch := TRUE;
   Fermi[1..6].V.WorkLimitSwitch := FALSE;
   Fermi[1..6].V.OilInPressure := FALSE;
   Fermi[1..6].V.Simulation := FALSE;
   Fermi[1..6].V.Config.RestLimSwitchExist := TRUE;
   Fermi[1..6].V.Config.WorkLimSwitchExist := FALSE;
   Fermi[1..6].V.Config.CheckOilInPressure := FALSE;
   Fermi[1..6].V.Config.CutRestWhenIsAtRest := TRUE;
   Fermi[1..6].V.Config.CutWorkWhenIsAtWork := TRUE;
   Fermi[1..6].V.Config.RestTime := T#2S;
   Fermi[1..6].V.Config.WorkTime := T#2S;
   Fermi[1..6].V.Config.RestTimeOut := T#4S;
   Fermi[1..6].V.Config.WorkTimeOut := T#4S;
   Fermi[1..6].V.ValveSts.AlarmPresence := FALSE;
   Fermi[1..6].V.ValveSts.RestPermit := TRUE;
   Fermi[1..6].V.ValveSts.RestInProgress := FALSE;
   Fermi[1..6].V.ValveSts.IsAtRest := TRUE;
   Fermi[1..6].V.ValveSts.WorkPermit := TRUE;
   Fermi[1..6].V.ValveSts.WorkInProgress := FALSE;
   Fermi[1..6].V.ValveSts.IsAtWork := FALSE;
   Fermi[1..6].V.ValveSts.StandStill := TRUE;
   Fermi[1..6].V.RestSolenoid := FALSE;
   Fermi[1..6].V.WorkSolenoid := FALSE;
   Fermi[1..6].V.ReqOilPressure := FALSE;
   Fermi[1..6].V.IsAtRest := TRUE;
   Fermi[1..6].V.IsAtWork := FALSE;
   Fermi[1..6].V.Ctrl.RestReq := FALSE;
   Fermi[1..6].V.Ctrl.WorkReq := FALSE;
   Fermi[1..6].V.Ctrl.RestSolenoid := FALSE;
   Fermi[1..6].V.Ctrl.WorkSolenoid := FALSE;
   Fermi[1..6].V.tonRest.PT := T#2S;
   Fermi[1..6].V.tonRest.IN := TRUE;
   Fermi[1..6].V.tonWork.PT := T#0MS;
   Fermi[1..6].V.tonWork.IN := FALSE;
   Fermi[1..6].V.tonTimeOutRest.PT := T#0MS;
   Fermi[1..6].V.tonTimeOutRest.IN := FALSE;
   Fermi[1..6].V.tonTimeOutWork.PT := T#0MS;
   Fermi[1..6].V.tonTimeOutWork.IN := FALSE;
   Fermi[1..6].TON_NoPendingCmd.PT := T#500MS;
   Fermi[1..6].TON_NoPendingCmd.IN := TRUE;
   Fermi[1..6].TON_Rest_MissingExtEnable.PT := T#0MS;
   Fermi[1..6].TON_Rest_MissingExtEnable.IN := FALSE;
   Fermi[1..6].TON_Work_MissingExtEnable.PT := T#0MS;
   Fermi[1..6].TON_Work_MissingExtEnable.IN := FALSE;
   Fermi[1..6].TON_PressureRunning_Timeout.PT := T#0MS;
   Fermi[1..6].TON_PressureRunning_Timeout.IN := FALSE;
   Fermi[1..6].Aux.Pb_Rest := FALSE;
   Fermi[1..6].Aux.Pb_Work := FALSE;
   Fermi[1..6].Aux.Pb_StartStop := FALSE;
   Pareggiatore.AreaInterface.EStop := FALSE;
   Pareggiatore.AreaInterface.Man := TRUE;
   Pareggiatore.AreaInterface.Aut := FALSE;
   Pareggiatore.AreaInterface.Cycle := FALSE;
   Pareggiatore.AreaInterface.StopInPhase := FALSE;
   Pareggiatore.AreaInterface.StopProgrammed := FALSE;
   Pareggiatore.AreaInterface.RstAlarms := FALSE;
   Pareggiatore.AreaInterface.ManOneShot := FALSE;
   Pareggiatore.AreaInterface.AutOneShot := FALSE;
   Pareggiatore.AreaInterface.CycleOneShot := FALSE;
   Pareggiatore.AreaInterface.CheckAutReady := FALSE;
   Pareggiatore.ZSI.Door_NormalStop := FALSE;
   Pareggiatore.ZSI.Door_SafeStop := FALSE;
   Pareggiatore.ZSI.Door_Opened := FALSE;
   Pareggiatore.ZSI.Door_EntryEnable := FALSE;
   Pareggiatore.DSI.SafeStop := FALSE;
   Pareggiatore.DSI.PowerEnable := TRUE;
   Pareggiatore.DSI.DevicesInSafeState := FALSE;
   Pareggiatore.DataIn.PB.Rest := FALSE;
   Pareggiatore.DataIn.PB.Work := FALSE;
   Pareggiatore.DataIn.PB.StartStop := FALSE;
   Pareggiatore.DataIn.Rest_Ls[1..8] := FALSE;
   Pareggiatore.DataIn.Work_Ls[1..8] := FALSE;
   Pareggiatore.Cin.Manager.EnableStopDoorOpeningReq := FALSE;
   Pareggiatore.Cin.Manager.EnableStopInPhase := FALSE;
   Pareggiatore.Cin.Manager.EnableStopProgrammed := FALSE;
   Pareggiatore.Cin.Manager.Control_ON := FALSE;
   Pareggiatore.Cin.Manager.Rest := FALSE;
   Pareggiatore.Cin.Manager.Work := FALSE;
   Pareggiatore.Cin.PressureRunning := FALSE;
   Pareggiatore.Cin.Rest_ExtEnable := TRUE;
   Pareggiatore.Cin.Work_ExtEnable := TRUE;
   Pareggiatore.Cin.ExternalAlarms := FALSE;
   Pareggiatore.Config.DelayPressureRunningTimeout := T#3S;
   Pareggiatore.Config.DelayMissingCondition := T#3S;
   Pareggiatore.Config.Rest_LsQty := 1;
   Pareggiatore.Config.Work_LsQty := 1;
   Pareggiatore.Config.Rest_RetainAut := FALSE;
   Pareggiatore.Config.Work_RetainAut := FALSE;
   Pareggiatore.Config.V.RestLimSwitchExist := TRUE;
   Pareggiatore.Config.V.WorkLimSwitchExist := TRUE;
   Pareggiatore.Config.V.CheckOilInPressure := FALSE;
   Pareggiatore.Config.V.CutRestWhenIsAtRest := TRUE;
   Pareggiatore.Config.V.CutWorkWhenIsAtWork := TRUE;
   Pareggiatore.Config.V.RestTime := T#1S;
   Pareggiatore.Config.V.WorkTime := T#1S;
   Pareggiatore.Config.V.RestTimeOut := T#1H;
   Pareggiatore.Config.V.WorkTimeOut := T#1H;
   Pareggiatore.MachineInterface.AutReady := FALSE;
   Pareggiatore.MachineInterface.Aborting := FALSE;
   Pareggiatore.MachineInterface.AckStopInPhase := FALSE;
   Pareggiatore.MachineInterface.AckStopProgrammed := FALSE;
   Pareggiatore.MachineInterface.MotionsStandStill := TRUE;
   Pareggiatore.MachineInterface.AlarmsPresence := FALSE;
   Pareggiatore.MachineInterface.WarningPresence := FALSE;
   Pareggiatore.COut.CtrlSafe := FALSE;
   Pareggiatore.COut.Standstill := TRUE;
   Pareggiatore.COut.ReqOilPressure := FALSE;
   Pareggiatore.COut.Rest_CheckNext := FALSE;
   Pareggiatore.COut.Work_CheckNext := FALSE;
   Pareggiatore.COut.Rest := FALSE;
   Pareggiatore.COut.Work := FALSE;
   Pareggiatore.DataOut.RestSolenoid := FALSE;
   Pareggiatore.DataOut.WorkSolenoid := FALSE;
   Pareggiatore.Sts.Standstill := TRUE;
   Pareggiatore.Sts.AlarmsPresence := FALSE;
   Pareggiatore.Sts.WarningsPresence := FALSE;
   Pareggiatore.Sts.Rest_Cnd := TRUE;
   Pareggiatore.Sts.Work_Cnd := TRUE;
   Pareggiatore.Ctrl.StopDueDoorOpeningRequest := FALSE;
   Pareggiatore.Ctrl.StopInPhase := FALSE;
   Pareggiatore.Ctrl.StopProgrammed := FALSE;
   Pareggiatore.Ctrl.StopAborting := FALSE;
   Pareggiatore.Ctrl.Work := FALSE;
   Pareggiatore.Ctrl.Rest := FALSE;
   Pareggiatore.Ctrl.Rest_Man := FALSE;
   Pareggiatore.Ctrl.Work_Man := FALSE;
   Pareggiatore.Ctrl.Rest_Aut := FALSE;
   Pareggiatore.Ctrl.Work_Aut := FALSE;
   Pareggiatore.V.ValveCtrl.SafeStop := FALSE;
   Pareggiatore.V.ValveCtrl.Rst := FALSE;
   Pareggiatore.V.ValveCtrl.MoveRest := FALSE;
   Pareggiatore.V.ValveCtrl.MoveWork := FALSE;
   Pareggiatore.V.RestLimitSwitch := FALSE;
   Pareggiatore.V.WorkLimitSwitch := FALSE;
   Pareggiatore.V.OilInPressure := FALSE;
   Pareggiatore.V.Simulation := FALSE;
   Pareggiatore.V.Config.RestLimSwitchExist := TRUE;
   Pareggiatore.V.Config.WorkLimSwitchExist := TRUE;
   Pareggiatore.V.Config.CheckOilInPressure := FALSE;
   Pareggiatore.V.Config.CutRestWhenIsAtRest := TRUE;
   Pareggiatore.V.Config.CutWorkWhenIsAtWork := TRUE;
   Pareggiatore.V.Config.RestTime := T#1S;
   Pareggiatore.V.Config.WorkTime := T#1S;
   Pareggiatore.V.Config.RestTimeOut := T#1H;
   Pareggiatore.V.Config.WorkTimeOut := T#1H;
   Pareggiatore.V.ValveSts.AlarmPresence := FALSE;
   Pareggiatore.V.ValveSts.RestPermit := TRUE;
   Pareggiatore.V.ValveSts.RestInProgress := FALSE;
   Pareggiatore.V.ValveSts.IsAtRest := FALSE;
   Pareggiatore.V.ValveSts.WorkPermit := TRUE;
   Pareggiatore.V.ValveSts.WorkInProgress := FALSE;
   Pareggiatore.V.ValveSts.IsAtWork := FALSE;
   Pareggiatore.V.ValveSts.StandStill := TRUE;
   Pareggiatore.V.RestSolenoid := FALSE;
   Pareggiatore.V.WorkSolenoid := FALSE;
   Pareggiatore.V.ReqOilPressure := FALSE;
   Pareggiatore.V.IsAtRest := FALSE;
   Pareggiatore.V.IsAtWork := FALSE;
   Pareggiatore.V.Ctrl.RestReq := FALSE;
   Pareggiatore.V.Ctrl.WorkReq := FALSE;
   Pareggiatore.V.Ctrl.RestSolenoid := FALSE;
   Pareggiatore.V.Ctrl.WorkSolenoid := FALSE;
   Pareggiatore.V.tonRest.PT := T#0MS;
   Pareggiatore.V.tonRest.IN := FALSE;
   Pareggiatore.V.tonWork.PT := T#0MS;
   Pareggiatore.V.tonWork.IN := FALSE;
   Pareggiatore.V.tonTimeOutRest.PT := T#0MS;
   Pareggiatore.V.tonTimeOutRest.IN := FALSE;
   Pareggiatore.V.tonTimeOutWork.PT := T#0MS;
   Pareggiatore.V.tonTimeOutWork.IN := FALSE;
   Pareggiatore.TON_NoPendingCmd.PT := T#500MS;
   Pareggiatore.TON_NoPendingCmd.IN := TRUE;
   Pareggiatore.TON_Rest_MissingExtEnable.PT := T#0MS;
   Pareggiatore.TON_Rest_MissingExtEnable.IN := FALSE;
   Pareggiatore.TON_Work_MissingExtEnable.PT := T#0MS;
   Pareggiatore.TON_Work_MissingExtEnable.IN := FALSE;
   Pareggiatore.TON_PressureRunning_Timeout.PT := T#0MS;
   Pareggiatore.TON_PressureRunning_Timeout.IN := FALSE;
   Pareggiatore.Aux.Pb_Rest := FALSE;
   Pareggiatore.Aux.Pb_Work := FALSE;
   Pareggiatore.Aux.Pb_StartStop := FALSE;
   TON_OP_REST_MissingCnd.PT := T#0MS;
   TON_OP_REST_MissingCnd.IN := FALSE;
   TON_OP_WORK_MissingCnd.PT := T#0MS;
   TON_OP_WORK_MissingCnd.IN := FALSE;
END_DATA_BLOCK

